DATA_BLOCK "PartErrorsCounter"   // DB46
{ S7_Optimized_Access := 'TRUE' }
VERSION : 0.1
// stored: AutoNumber true, DBAccessibleFromOPCUA true, DBAccessibleFromWebserver true, IsOnlyStoredInLoadMemory false, IsRetainMemResEnabled false, IsWriteProtectedInAS false, MemoryReserve 100
   VAR RETAIN
      CountersRef { S7_SetPoint := 'True'} : Array[1.."NumberOfProductionPrograms"] of "UDT_NOKcounter";
   END_VAR
   VAR
      CountersHMI : "UDT_NOKcounter";
   END_VAR
BEGIN
   CountersRef[1].Counters[0,0..50] := 0;
   CountersRef[1].Counters[1,0..9] := 0;
   CountersRef[1].Counters[1,10] := 2;
   CountersRef[1].Counters[1,11] := 1;
   CountersRef[1].Counters[1,12..19] := 0;
   CountersRef[1].Counters[1,20] := 3;
   CountersRef[1].Counters[1,21] := 1;
   CountersRef[1].Counters[1,22..33] := 0;
   CountersRef[1].Counters[1,34] := 1;
   CountersRef[1].Counters[1,35..43] := 0;
   CountersRef[1].Counters[1,44] := 1;
   CountersRef[1].Counters[1,45..50] := 0;
   CountersRef[1].Counters[2,0..13] := 0;
   CountersRef[1].Counters[2,14] := 1;
   CountersRef[1].Counters[2,15..20] := 0;
   CountersRef[1].Counters[2,21] := 1;
   CountersRef[1].Counters[2,22..50] := 0;
   CountersRef[1].Counters[3,0..50] := 0;
   CountersRef[2].Counters[0,0..50] := 0;
   CountersRef[2].Counters[1,0..9] := 0;
   CountersRef[2].Counters[1,10] := 4;
   CountersRef[2].Counters[1,11] := 1;
   CountersRef[2].Counters[1,12..19] := 0;
   CountersRef[2].Counters[1,20] := 3;
   CountersRef[2].Counters[1,21] := 2;
   CountersRef[2].Counters[1,22..50] := 0;
   CountersRef[2].Counters[2,0..10] := 0;
   CountersRef[2].Counters[2,11] := 1;
   CountersRef[2].Counters[2,12..13] := 0;
   CountersRef[2].Counters[2,14] := 1;
   CountersRef[2].Counters[2,15..20] := 0;
   CountersRef[2].Counters[2,21] := 1;
   CountersRef[2].Counters[2,22..23] := 0;
   CountersRef[2].Counters[2,24] := 1;
   CountersRef[2].Counters[2,25..30] := 0;
   CountersRef[2].Counters[2,31] := 1;
   CountersRef[2].Counters[2,32..33] := 0;
   CountersRef[2].Counters[2,34] := 1;
   CountersRef[2].Counters[2,35..40] := 0;
   CountersRef[2].Counters[2,41] := 1;
   CountersRef[2].Counters[2,42..43] := 0;
   CountersRef[2].Counters[2,44] := 1;
   CountersRef[2].Counters[2,45..50] := 0;
   CountersRef[2].Counters[3,0..50] := 0;
   CountersRef[3].Counters[0,0..50] := 0;
   CountersRef[3].Counters[1,0..50] := 0;
   CountersRef[3].Counters[2,0..50] := 0;
   CountersRef[3].Counters[3,0..50] := 0;
   CountersRef[4].Counters[0,0..50] := 0;
   CountersRef[4].Counters[1,0..50] := 0;
   CountersRef[4].Counters[2,0..50] := 0;
   CountersRef[4].Counters[3,0..50] := 0;
   CountersRef[5].Counters[0,0..50] := 0;
   CountersRef[5].Counters[1,0..9] := 0;
   CountersRef[5].Counters[1,10] := 17;
   CountersRef[5].Counters[1,11] := 6;
   CountersRef[5].Counters[1,12..19] := 0;
   CountersRef[5].Counters[1,20..21] := 1;
   CountersRef[5].Counters[1,22..50] := 0;
   CountersRef[5].Counters[2,0..9] := 0;
   CountersRef[5].Counters[2,10] := 4;
   CountersRef[5].Counters[2,11] := 3;
   CountersRef[5].Counters[2,12..13] := 0;
   CountersRef[5].Counters[2,14] := 1;
   CountersRef[5].Counters[2,15..23] := 0;
   CountersRef[5].Counters[2,24] := 4;
   CountersRef[5].Counters[2,25..50] := 0;
   CountersRef[5].Counters[3,0..50] := 0;
   CountersRef[6].Counters[0,0..50] := 0;
   CountersRef[6].Counters[1,0..50] := 0;
   CountersRef[6].Counters[2,0..9] := 0;
   CountersRef[6].Counters[2,10] := 1;
   CountersRef[6].Counters[2,11..13] := 0;
   CountersRef[6].Counters[2,14] := 1;
   CountersRef[6].Counters[2,15..21] := 0;
   CountersRef[6].Counters[2,22] := 1;
   CountersRef[6].Counters[2,23..33] := 0;
   CountersRef[6].Counters[2,34] := 2;
   CountersRef[6].Counters[2,35..43] := 0;
   CountersRef[6].Counters[2,44] := 2;
   CountersRef[6].Counters[2,45..50] := 0;
   CountersRef[6].Counters[3,0..50] := 0;
   CountersRef[7].Counters[0,0..50] := 0;
   CountersRef[7].Counters[1,0..50] := 0;
   CountersRef[7].Counters[2,0..50] := 0;
   CountersRef[7].Counters[3,0..50] := 0;
   CountersRef[8].Counters[0,0..50] := 0;
   CountersRef[8].Counters[1,0..50] := 0;
   CountersRef[8].Counters[2,0..50] := 0;
   CountersRef[8].Counters[3,0..50] := 0;
   CountersHMI.Counters[0,0..50] := 0;
   CountersHMI.Counters[1,0..50] := 0;
   CountersHMI.Counters[2,0..50] := 0;
   CountersHMI.Counters[3,0..50] := 0;
END_DATA_BLOCK

DATA_BLOCK "READER_MODEL"   // DB74
{ S7_Optimized_Access := 'TRUE' }
VERSION : 0.1
// stored: AutoNumber true, DBAccessibleFromOPCUA true, DBAccessibleFromWebserver true, IsOnlyStoredInLoadMemory false, IsRetainMemResEnabled false, IsWriteProtectedInAS false, MemoryReserve 100
   VAR RETAIN
      PRODUCT { S7_SetPoint := 'True'} : Array[0.."NumberOfProductionPrograms"] of "READER_PRODUCT";
   END_VAR
BEGIN
   PRODUCT[1..4].SIDE_RH.POSITION := 13;
   PRODUCT[1..4].SIDE_RH.LEN := 3;
   PRODUCT[1].SIDE_RH.STRING_LABEL := '336';
   PRODUCT[2].SIDE_RH.STRING_LABEL := '532';
   PRODUCT[3].SIDE_RH.STRING_LABEL := '336';
   PRODUCT[4].SIDE_RH.STRING_LABEL := '532';
   PRODUCT[1..4].SIDE_RH.READER_BYPASS := FALSE;
   PRODUCT[1..4].SIDE_LH.POSITION := 13;
   PRODUCT[1..4].SIDE_LH.LEN := 3;
   PRODUCT[1].SIDE_LH.STRING_LABEL := '328';
   PRODUCT[2].SIDE_LH.STRING_LABEL := '526';
   PRODUCT[3].SIDE_LH.STRING_LABEL := '328';
   PRODUCT[4].SIDE_LH.STRING_LABEL := '526';
   PRODUCT[1..4].SIDE_LH.READER_BYPASS := FALSE;
   PRODUCT[1..4].REAR_TUBE.POSITION := 13;
   PRODUCT[1..4].REAR_TUBE.LEN := 3;
   PRODUCT[1].REAR_TUBE.STRING_LABEL := '343';
   PRODUCT[2].REAR_TUBE.STRING_LABEL := '514';
   PRODUCT[3].REAR_TUBE.STRING_LABEL := '343';
   PRODUCT[4].REAR_TUBE.STRING_LABEL := '514';
   PRODUCT[1..4].REAR_TUBE.READER_BYPASS := FALSE;
   PRODUCT[1..2].FRONT_TUBE.POSITION := 13;
   PRODUCT[1..2].FRONT_TUBE.LEN := 3;
   PRODUCT[1..2].FRONT_TUBE.STRING_LABEL := '907';
   PRODUCT[1..4].FRONT_TUBE.READER_BYPASS := TRUE;
   PRODUCT[1..2].NUM_TUBE := TRUE;
   PRODUCT[3].NUM_TUBE := FALSE;
END_DATA_BLOCK

DATA_BLOCK "READER_MODEL_ACTUAL"   // DB75
{ S7_Optimized_Access := 'TRUE' }
VERSION : 0.1
// stored: AutoNumber true, DBAccessibleFromOPCUA true, DBAccessibleFromWebserver true, IsOnlyStoredInLoadMemory false, IsRetainMemResEnabled false, IsWriteProtectedInAS false, MemoryReserve 100
   VAR
      PRODUCTO : "READER_PRODUCT";
      ST1_TABLE_1 : Struct
         SIDE_RH : String;
         SIDE_LH : String;
         REAR_TUBE : String;
         FRONT_TUBE : String;
         NFP_AUX : String;
      END_STRUCT;
      ST2_TABLE_2 : Struct
         SIDE_RH : String;
         SIDE_LH : String;
         REAR_TUBE : String;
         FRONT_TUBE : String;
         NFP_AUX : String;
      END_STRUCT;
      ST3_FITTING : Struct
         SIDE_RH : String;
         SIDE_LH : String;
         REAR_TUBE : String;
         FRONT_TUBE : String;
         NFP_AUX : String;
      END_STRUCT;
      R1_GRIPPER : Struct
         SIDE_RH : String;
         SIDE_LH : String;
         REAR_TUBE : String;
         FRONT_TUBE : String;
         NFP_AUX : String;
      END_STRUCT;
      R2_GRIPPER : Struct
         SIDE_RH : String;
         SIDE_LH : String;
         REAR_TUBE : String;
         FRONT_TUBE : String;
         NFP_AUX : String;
      END_STRUCT;
      ALL_SCANNER_OK : Bool;
      SIDE_LH_SCANNER_OK : Bool;
      SIDE_RH_SCANNER_OK : Bool;
      REAR_TUBE_SCANNER_OK : Bool;
      FRONT_TUBE_SCANNER_OK : Bool;
      IN_BOX : "READER_PRODUCT";
      EDIT : "READER_PRODUCT";
      READER { S7_SetPoint := 'True'} : String;
      ST_CLEAR : Struct
         SIDE_RH : String;
         SIDE_LH : String;
         REAR_TUBE : String;
         FRONT_TUBE : String;
         NFP_AUX : String;
      END_STRUCT;
      SCAN_CLEAR : Bool;
      RECIBIDO_ESCANER_REAR_TUBE : Array[0..254] of Char;
      RECIBIDO_ESCANER_FRONT_TUBE : Array[0..254] of Char;
      RECIBIDO_ESCANER_RH_MEMBER : Array[0..254] of Char;
      RECIBIDO_ESCANER_LH_MEMBER : Array[0..254] of Char;
      RECIBIDO_ESCANER_REAR_TUBE_STRING : String;
      RECIBIDO_ESCANER_FRONT_TUBE_STRING : String;
      RECIBIDO_ESCANER_RH_MEMBER_STRING : String;
      RECIBIDO_ESCANER_LH_MEMBER_STRING : String;
      LECTURA_ESCANER_REAR_TUBE : String;
      LECTURA_ESCANER_FRONT_TUBE : String;
      LECTURA_ESCANER_RH_MEMBER : String;
      LECTURA_ESCANER_LH_MEMBER : String;
   END_VAR
BEGIN
END_DATA_BLOCK

DATA_BLOCK "MII_Interface_Configuration"   // DB2021
{ S7_Optimized_Access := 'TRUE' }
VERSION : 0.1
// stored: AutoNumber false, DBAccessibleFromOPCUA true, DBAccessibleFromWebserver true, IsOnlyStoredInLoadMemory false, IsRetainMemResEnabled false, IsWriteProtectedInAS false, MemoryReserve 100
   VAR
      Connection { ExternalAccessible := 'False'; ExternalVisible := 'False'; ExternalWritable := 'False'} : Struct
         ConnectInfo { ExternalAccessible := 'False'; ExternalVisible := 'False'; ExternalWritable := 'False'; S7_SetPoint := 'True'} : OPC_UA_SessionConnectInfo;
         ConnectionHdl { ExternalAccessible := 'False'; ExternalVisible := 'False'; ExternalWritable := 'False'} : DWord;
         ServerEndpointUrl { ExternalAccessible := 'False'; ExternalVisible := 'False'; ExternalWritable := 'False'} : String[254] := 'opc.tcp://:4840';
      END_STRUCT;
      Namespaces { ExternalAccessible := 'False'; ExternalVisible := 'False'; ExternalWritable := 'False'} : Struct
         NamespaceURIs { ExternalAccessible := 'False'; ExternalVisible := 'False'; ExternalWritable := 'False'} : Array[0..0] of WString;
         ServerNamespaceIndexes { ExternalAccessible := 'False'; ExternalVisible := 'False'; ExternalWritable := 'False'} : Array[0..0] of UInt;
         NamespaceStatusList { ExternalAccessible := 'False'; ExternalVisible := 'False'; ExternalWritable := 'False'} : Array[0..0] of DWord;
         NamespaceCount { ExternalAccessible := 'False'; ExternalVisible := 'False'; ExternalWritable := 'False'} : UInt := 1;
      END_STRUCT;
      MethodLists { ExternalAccessible := 'False'; ExternalVisible := 'False'; ExternalWritable := 'False'} : Struct
         MII_METHODS { ExternalAccessible := 'False'; ExternalVisible := 'False'; ExternalWritable := 'False'} : Struct
            MethodCount { ExternalAccessible := 'False'; ExternalVisible := 'False'; ExternalWritable := 'False'} : UInt := 9;
            ObjectNodes { ExternalAccessible := 'False'; ExternalVisible := 'False'; ExternalWritable := 'False'; S7_SetPoint := 'True'} : Array[0..8] of OPC_UA_NodeId;
            MethodNodes { ExternalAccessible := 'False'; ExternalVisible := 'False'; ExternalWritable := 'False'; S7_SetPoint := 'True'} : Array[0..8] of OPC_UA_NodeId;
            MethodHdls { ExternalAccessible := 'False'; ExternalVisible := 'False'; ExternalWritable := 'False'} : Array[0..8] of DWord;
         END_STRUCT;
      END_STRUCT;
   END_VAR
BEGIN
   Connection.ConnectInfo.SessionName := WSTRING#'OPC UA Connection_1';
   Connection.ConnectInfo.ApplicationName := WSTRING#'';
   Connection.ConnectInfo.SecurityMsgMode := 1;
   Connection.ConnectInfo.SecurityPolicy := 1;
   Connection.ConnectInfo.CheckServerCertificate := False;
   Connection.ConnectInfo.TransportProfile := 1;
   Connection.ConnectInfo.UserIdentityTokenType := 0;
   Connection.ConnectInfo.CertificateID := 0;
   Connection.ConnectInfo.SessionTimeout := T#30S;
   Connection.ConnectInfo.MonitorConnection := T#5S;
   Connection.ConnectInfo.LocaleIDs[0] := 'en-US';
   Connection.ConnectInfo.LocaleIDs[1..4] := '';
   Namespaces.NamespaceURIs[0] := WSTRING#'http://sap.com/PCoUaServer/Destinations';
   MethodLists.MII_METHODS.ObjectNodes[0..8].NamespaceIndex := 0;
   MethodLists.MII_METHODS.ObjectNodes[0..8].Identifier := WSTRING#'a72e725d-6be7-4a17-bcd4-0be67b6cbfbe';
   MethodLists.MII_METHODS.ObjectNodes[0..8].IdentifierType := 1;
   MethodLists.MII_METHODS.MethodNodes[0..8].NamespaceIndex := 0;
   MethodLists.MII_METHODS.MethodNodes[0].Identifier := WSTRING#'5e83d9d8-abe4-4ece-894f-119f40c23d1f';
   MethodLists.MII_METHODS.MethodNodes[1].Identifier := WSTRING#'3a6a30a3-a9b9-4f00-ac48-5dfb28f8e6a4';
   MethodLists.MII_METHODS.MethodNodes[2].Identifier := WSTRING#'fc62dbc1-f795-4566-bb4d-0b596c22b389';
   MethodLists.MII_METHODS.MethodNodes[3].Identifier := WSTRING#'c66a08a9-d6b4-453f-b0e9-0d4ff2f595c1';
   MethodLists.MII_METHODS.MethodNodes[4].Identifier := WSTRING#'a12cda35-f7c0-4943-b30d-d26694925508';
   MethodLists.MII_METHODS.MethodNodes[5].Identifier := WSTRING#'9febe458-2cc0-4c91-b17b-56067f98920d';
   MethodLists.MII_METHODS.MethodNodes[6].Identifier := WSTRING#'9fd0466f-1121-4821-944e-2d89fa189b19';
   MethodLists.MII_METHODS.MethodNodes[7].Identifier := WSTRING#'1a97343a-fec3-434f-bd32-25d77a49b705';
   MethodLists.MII_METHODS.MethodNodes[8].Identifier := WSTRING#'d0a2f4c1-2dea-442d-aa14-aa44dfe57828';
   MethodLists.MII_METHODS.MethodNodes[0..8].IdentifierType := 1;
END_DATA_BLOCK

DATA_BLOCK "MII_Interface_Data"   // DB2022
{ S7_Optimized_Access := 'TRUE' }
VERSION : 0.1
// stored: AutoNumber false, DBAccessibleFromOPCUA true, DBAccessibleFromWebserver true, IsOnlyStoredInLoadMemory false, IsRetainMemResEnabled false, IsWriteProtectedInAS false, MemoryReserve 100
   VAR
      MII_METHODS { ExternalAccessible := 'False'; ExternalVisible := 'False'; ExternalWritable := 'False'} : Struct
         MethodStatusList { ExternalAccessible := 'False'; ExternalVisible := 'False'; ExternalWritable := 'False'} : Array[0..8] of DWord;
         MethodResultList { ExternalAccessible := 'False'; ExternalVisible := 'False'; ExternalWritable := 'False'} : Array[0..8] of DWord;
         M000_PRODUCTION_DECLARATION { ExternalAccessible := 'False'; ExternalVisible := 'False'; ExternalWritable := 'False'} : Struct
            Inputs { ExternalAccessible := 'False'; ExternalVisible := 'False'; ExternalWritable := 'False'; S7_SetPoint := 'True'} : "MII_Interface.MII_METHODS.M000_PRODUCTION_DECLARATION.Inputs";   // the definition of the input argument of method 1:Destinations.1:PRODUCTION_DECLARATION
            Outputs { ExternalAccessible := 'False'; ExternalVisible := 'False'; ExternalWritable := 'False'; S7_SetPoint := 'True'} : "MII_Interface.MII_METHODS.M000_PRODUCTION_DECLARATION.Outputs";   // the definition of the output arguments of method 1:Destinations.1:PRODUCTION_DECLARATION
         END_STRUCT;
         M001_GET_LOCAL_TIME { ExternalAccessible := 'False'; ExternalVisible := 'False'; ExternalWritable := 'False'} : Struct
            Outputs { ExternalAccessible := 'False'; ExternalVisible := 'False'; ExternalWritable := 'False'; S7_SetPoint := 'True'} : "MII_Interface.MII_METHODS.M001_GET_LOCAL_TIME.Outputs";   // the definition of the output arguments of method 2:Destinations.2:2_GET_LOCAL_TIME
         END_STRUCT;
         M101_SCRAP_DECLARATION { ExternalAccessible := 'False'; ExternalVisible := 'False'; ExternalWritable := 'False'} : Struct
            Inputs { ExternalAccessible := 'False'; ExternalVisible := 'False'; ExternalWritable := 'False'; S7_SetPoint := 'True'} : "MII_Interface.MII_METHODS.M101_SCRAP_DECLARATION.Inputs";   // the definition of the input argument of method 2:Destinations.2:1_SCRAP_DECLARATION
            Outputs { ExternalAccessible := 'False'; ExternalVisible := 'False'; ExternalWritable := 'False'; S7_SetPoint := 'True'} : "MII_Interface.MII_METHODS.M101_SCRAP_DECLARATION.Outputs";   // the definition of the output arguments of method 2:Destinations.2:1_SCRAP_DECLARATION
         END_STRUCT;
         M003_GENERATE_ALERT { ExternalAccessible := 'False'; ExternalVisible := 'False'; ExternalWritable := 'False'} : Struct
            Inputs { ExternalAccessible := 'False'; ExternalVisible := 'False'; ExternalWritable := 'False'; S7_SetPoint := 'True'} : "MII_Interface.MII_METHODS.M003_GENERATE_ALERT.Inputs";   // the definition of the input argument of method 2:Destinations.2:3_GENERATE_ALERT
            Outputs { ExternalAccessible := 'False'; ExternalVisible := 'False'; ExternalWritable := 'False'; S7_SetPoint := 'True'} : "MII_Interface.MII_METHODS.M003_GENERATE_ALERT.Outputs";   // the definition of the output arguments of method 2:Destinations.2:3_GENERATE_ALERT
         END_STRUCT;
         M102_REWORK_DECLARATION { ExternalAccessible := 'False'; ExternalVisible := 'False'; ExternalWritable := 'False'} : Struct
            Inputs { ExternalAccessible := 'False'; ExternalVisible := 'False'; ExternalWritable := 'False'; S7_SetPoint := 'True'} : "MII_Interface.MII_METHODS.M102_REWORK_DECLARATION.Inputs";   // the definition of the input argument of method 2:Destinations.2:4_REWORK_DECLARATION
            Outputs { ExternalAccessible := 'False'; ExternalVisible := 'False'; ExternalWritable := 'False'; S7_SetPoint := 'True'} : "MII_Interface.MII_METHODS.M102_REWORK_DECLARATION.Outputs";   // the definition of the output arguments of method 2:Destinations.2:4_REWORK_DECLARATION
         END_STRUCT;
         M002_GET_PLANTS { ExternalAccessible := 'False'; ExternalVisible := 'False'; ExternalWritable := 'False'} : Struct
            Outputs { ExternalAccessible := 'False'; ExternalVisible := 'False'; ExternalWritable := 'False'; S7_SetPoint := 'True'} : "MII_Interface.MII_METHODS.M002_GET_PLANTS.Outputs";   // the definition of the output arguments of method 2:Destinations.2:M005_GET_PLANTS
         END_STRUCT;
         M004_NTRS { ExternalAccessible := 'False'; ExternalVisible := 'False'; ExternalWritable := 'False'} : Struct
            Inputs { ExternalAccessible := 'False'; ExternalVisible := 'False'; ExternalWritable := 'False'; S7_SetPoint := 'True'} : "MII_Interface.MII_METHODS.M004_NTRS.Inputs";   // the definition of the input argument of method 2:Destinations.2:M006_NTRS
            Outputs { ExternalAccessible := 'False'; ExternalVisible := 'False'; ExternalWritable := 'False'; S7_SetPoint := 'True'} : "MII_Interface.MII_METHODS.M004_NTRS.Outputs";   // the definition of the output arguments of method 2:Destinations.2:M006_NTRS
         END_STRUCT;
         M103_PY { ExternalAccessible := 'False'; ExternalVisible := 'False'; ExternalWritable := 'False'} : Struct
            Inputs { ExternalAccessible := 'False'; ExternalVisible := 'False'; ExternalWritable := 'False'; S7_SetPoint := 'True'} : "MII_Interface.MII_METHODS.M103_PY.Inputs";   // the definition of the input argument of method 2:Destinations.2:M103_PY
            Outputs { ExternalAccessible := 'False'; ExternalVisible := 'False'; ExternalWritable := 'False'; S7_SetPoint := 'True'} : "MII_Interface.MII_METHODS.M103_PY.Outputs";   // the definition of the output arguments of method 2:Destinations.2:M103_PY
         END_STRUCT;
         M005_VARIABILITY { ExternalAccessible := 'False'; ExternalVisible := 'False'; ExternalWritable := 'False'} : Struct
            Inputs { ExternalAccessible := 'False'; ExternalVisible := 'False'; ExternalWritable := 'False'; S7_SetPoint := 'True'} : "MII_Interface.MII_METHODS.M005_VARIABILITY.Inputs";   // the definition of the input argument of method 2:Destinations.2:M005_VARIABILITY
            Outputs { ExternalAccessible := 'False'; ExternalVisible := 'False'; ExternalWritable := 'False'; S7_SetPoint := 'True'} : "MII_Interface.MII_METHODS.M005_VARIABILITY.Outputs";   // the definition of the output arguments of method 2:Destinations.2:M005_VARIABILITY
         END_STRUCT;
      END_STRUCT;
   END_VAR
BEGIN
END_DATA_BLOCK

ORGANIZATION_BLOCK "OB_ProgramCycle"   // OB1, LAD, ProgramCycle
TITLE = "Main Program Sweep (Cycle)"
{ S7_Optimized_Access := 'TRUE' }
VERSION : 0.1
// stored: AutoNumber true, IsIECCheckEnabled false, SetENOAutomatically false
   VAR_INPUT
      Initial_Call : Bool;   // Initial call of this OB
      Remanence : Bool;   // =True, if remanent data are available
   END_VAR
   VAR_TEMP   // added for the SCL form of the ladder/FBD networks
      _w1 : Bool;
      _s5time1 : S5Time;
   END_VAR
BEGIN

REGION Network 1
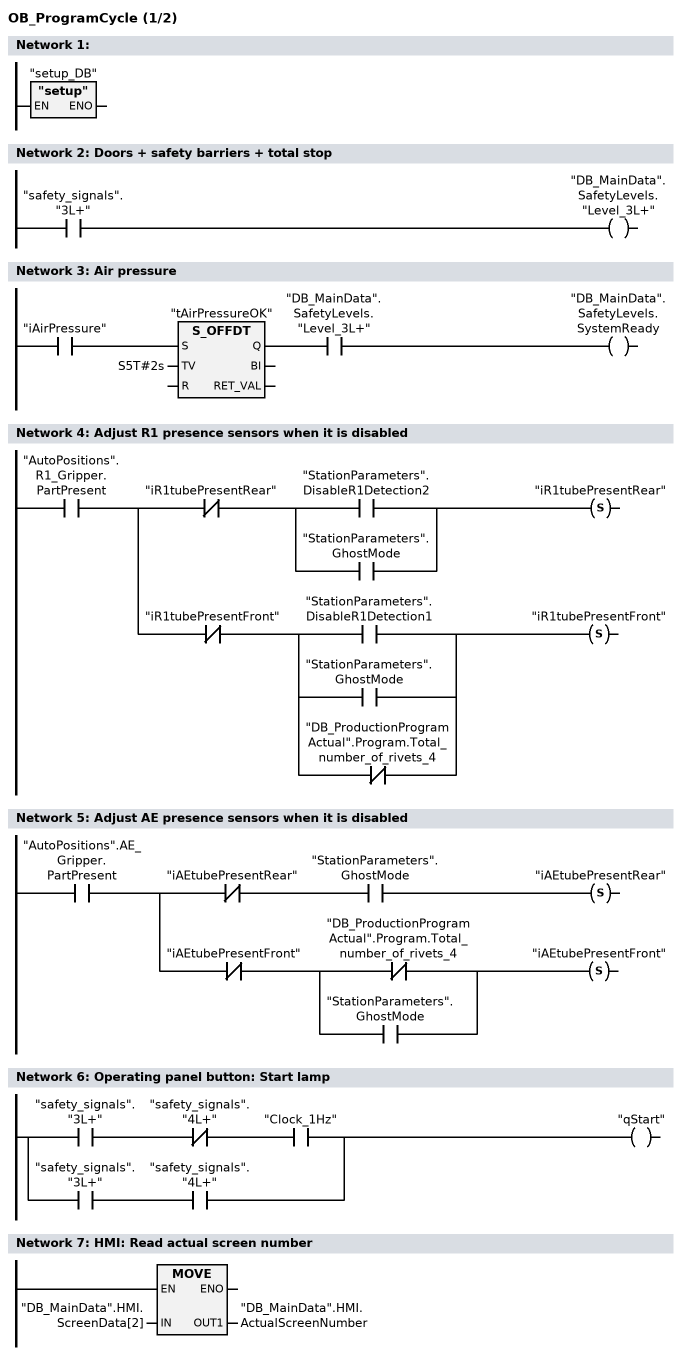
   RUNG wire#powerrail
      "setup_DB"()
   END_RUNG
   // the same network as SCL:
   "setup_DB"();   // "setup"
END_REGION

REGION Network 2: Doors + safety barriers + total stop
   RUNG wire#powerrail
      Contact( "safety_signals"."3L+" )
      Coil( "DB_MainData".SafetyLevels."Level_3L+" )
   END_RUNG
   // the same network as SCL:
   "DB_MainData".SafetyLevels."Level_3L+" := "safety_signals"."3L+";
END_REGION

REGION Network 3: Air pressure
   RUNG wire#powerrail
      Contact( "iAirPressure" )
      S_OFFDT(T_NO := "tAirPressureOK", TV := S5T#2s, R :=, BI =>, RET_VAL =>)
      Contact( "DB_MainData".SafetyLevels."Level_3L+" )
      Coil( "DB_MainData".SafetyLevels.SystemReady )
   END_RUNG
   // the same network as SCL:
   #_s5time1 := S_OFFDT(T_NO := "tAirPressureOK", S := "iAirPressure", TV := S5T#2s, Q => #_w1);
   "DB_MainData".SafetyLevels.SystemReady := #_w1 AND "DB_MainData".SafetyLevels."Level_3L+";
END_REGION

REGION Network 4: Adjust R1 presence sensors when it is disabled
   RUNG wire#powerrail
      Contact( "AutoPositions".R1_Gripper.PartPresent )
      wire#w1
      I_Contact( "iR1tubePresentRear" )
      wire#w2
      Contact( "StationParameters".DisableR1Detection2 )
      wire#w3
      S_Coil( "iR1tubePresentRear" )
   END_RUNG
   RUNG wire#w2
      Contact( "StationParameters".GhostMode )
   END_RUNG wire#w3
   RUNG wire#w1
      I_Contact( "iR1tubePresentFront" )
      wire#w4
      Contact( "StationParameters".DisableR1Detection1 )
      wire#w5
      S_Coil( "iR1tubePresentFront" )
   END_RUNG
   RUNG wire#w4
      Contact( "StationParameters".GhostMode )
   END_RUNG wire#w5
   RUNG wire#w4
      I_Contact( "DB_ProductionProgramActual".Program.Total_number_of_rivets_4 )
   END_RUNG wire#w5
   // the same network as SCL:
   IF "AutoPositions".R1_Gripper.PartPresent AND NOT "iR1tubePresentRear" AND ("StationParameters".DisableR1Detection2 OR "StationParameters".GhostMode) THEN
       "iR1tubePresentRear" := TRUE;
   END_IF;
   IF "AutoPositions".R1_Gripper.PartPresent AND NOT "iR1tubePresentFront" AND ("StationParameters".DisableR1Detection1 OR "StationParameters".GhostMode OR NOT "DB_ProductionProgramActual".Program.Total_number_of_rivets_4) THEN
       "iR1tubePresentFront" := TRUE;
   END_IF;
END_REGION

REGION Network 5: Adjust AE presence sensors when it is disabled
   RUNG wire#powerrail
      Contact( "AutoPositions".AE_Gripper.PartPresent )
      wire#w1
      I_Contact( "iAEtubePresentRear" )
      Contact( "StationParameters".GhostMode )
      S_Coil( "iAEtubePresentRear" )
   END_RUNG
   RUNG wire#w1
      I_Contact( "iAEtubePresentFront" )
      wire#w2
      I_Contact( "DB_ProductionProgramActual".Program.Total_number_of_rivets_4 )
      wire#w3
      S_Coil( "iAEtubePresentFront" )
   END_RUNG
   RUNG wire#w2
      Contact( "StationParameters".GhostMode )
   END_RUNG wire#w3
   // the same network as SCL:
   IF "AutoPositions".AE_Gripper.PartPresent AND NOT "iAEtubePresentRear" AND "StationParameters".GhostMode THEN
       "iAEtubePresentRear" := TRUE;
   END_IF;
   IF "AutoPositions".AE_Gripper.PartPresent AND NOT "iAEtubePresentFront" AND (NOT "DB_ProductionProgramActual".Program.Total_number_of_rivets_4 OR "StationParameters".GhostMode) THEN
       "iAEtubePresentFront" := TRUE;
   END_IF;
END_REGION

REGION Network 6: Operating panel button: Start lamp
   RUNG wire#powerrail
      Contact( "safety_signals"."3L+" )
      I_Contact( "safety_signals"."4L+" )
      Contact( "Clock_1Hz" )
      wire#w1
      Coil( "qStart" )
   END_RUNG
   RUNG wire#powerrail
      Contact( "safety_signals"."3L+" )
      Contact( "safety_signals"."4L+" )
   END_RUNG wire#w1
   // the same network as SCL:
   "qStart" := ("safety_signals"."3L+" AND NOT "safety_signals"."4L+" AND "Clock_1Hz") OR ("safety_signals"."3L+" AND "safety_signals"."4L+");
END_REGION

REGION Network 7: HMI: Read actual screen number
   RUNG wire#powerrail
      Move(in := "DB_MainData".HMI.ScreenData[2], out1 => "DB_MainData".HMI.ActualScreenNumber)
   END_RUNG
   // the same network as SCL:
   "DB_MainData".HMI.ActualScreenNumber := "DB_MainData".HMI.ScreenData[2];
END_REGION

REGION Network 8: FB_Main
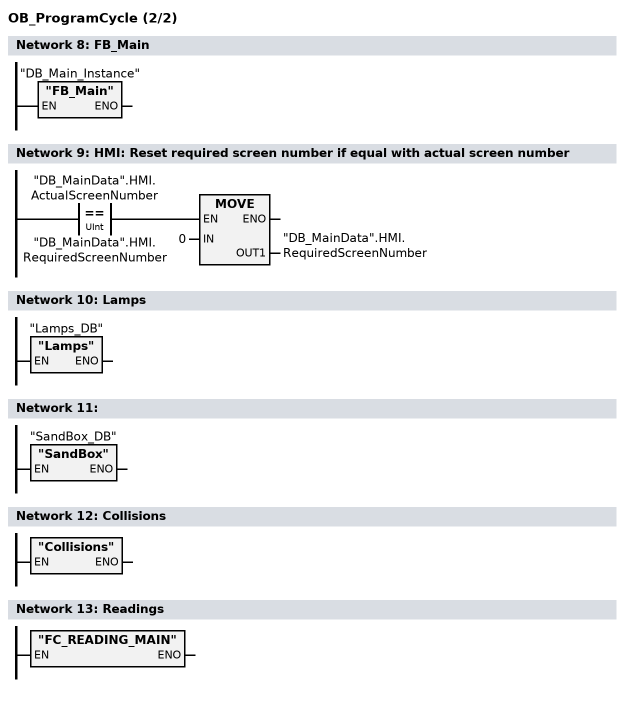
   RUNG wire#powerrail
      "DB_Main_Instance"()
   END_RUNG
   // the same network as SCL:
   "DB_Main_Instance"();   // "FB_Main"
END_REGION

REGION Network 9: HMI: Reset required screen number if equal with actual screen number
   RUNG wire#powerrail
      { S7_Templates := "SrcType := UInt" } EQ_Contact(in1 := "DB_MainData".HMI.ActualScreenNumber, in2 := "DB_MainData".HMI.RequiredScreenNumber)
      Move(in := 0, out1 => "DB_MainData".HMI.RequiredScreenNumber)
   END_RUNG
   // the same network as SCL:
   IF "DB_MainData".HMI.ActualScreenNumber = "DB_MainData".HMI.RequiredScreenNumber THEN
       "DB_MainData".HMI.RequiredScreenNumber := 0;
   END_IF;
END_REGION

REGION Network 10: Lamps
   RUNG wire#powerrail
      "Lamps_DB"()
   END_RUNG
   // the same network as SCL:
   "Lamps_DB"();   // "Lamps"
END_REGION

REGION Network 11
   RUNG wire#powerrail
      "SandBox_DB"()
   END_RUNG
   // the same network as SCL:
   "SandBox_DB"();   // "SandBox"
END_REGION

REGION Network 12: Collisions
   RUNG wire#powerrail
      "Collisions"()
   END_RUNG
   // the same network as SCL:
   "Collisions"();
END_REGION

REGION Network 13: Readings
   RUNG wire#powerrail
      "FC_READING_MAIN"()
   END_RUNG
   // the same network as SCL:
   "FC_READING_MAIN"();
END_REGION
END_ORGANIZATION_BLOCK

FUNCTION_BLOCK "FB_Main"   // FB5000, LAD
{ S7_Optimized_Access := 'TRUE' }
VERSION : 0.1
// stored: AutoNumber false, IsIECCheckEnabled false, IsRetainMemResEnabled false, MemoryReserve 100, SetENOAutomatically false, UDAEnableTagReadback false
   VAR
      IEC_Timer_0_Instance { S7_SetPoint := 'True'} : TON_TIME;
      MachineModeOld { S7_SetPoint := 'True'} : UInt;
      F_TRIG_Instance { S7_SetPoint := 'True'} : F_TRIG;
      F_TRIG_Instance_1 { S7_SetPoint := 'True'} : F_TRIG;
      F_TRIG_Instance_2 { S7_SetPoint := 'True'} : F_TRIG;
      R_TRIG_Instance { S7_SetPoint := 'True'} : R_TRIG;
      R_TRIG_Instance_1 { S7_SetPoint := 'True'} : R_TRIG;
   END_VAR
   VAR_TEMP   // added for the SCL form of the ladder/FBD networks
      _w1 : Bool;
      _w2 : Bool;
   END_VAR
BEGIN

REGION Network 1: alarms fc, lamp fc
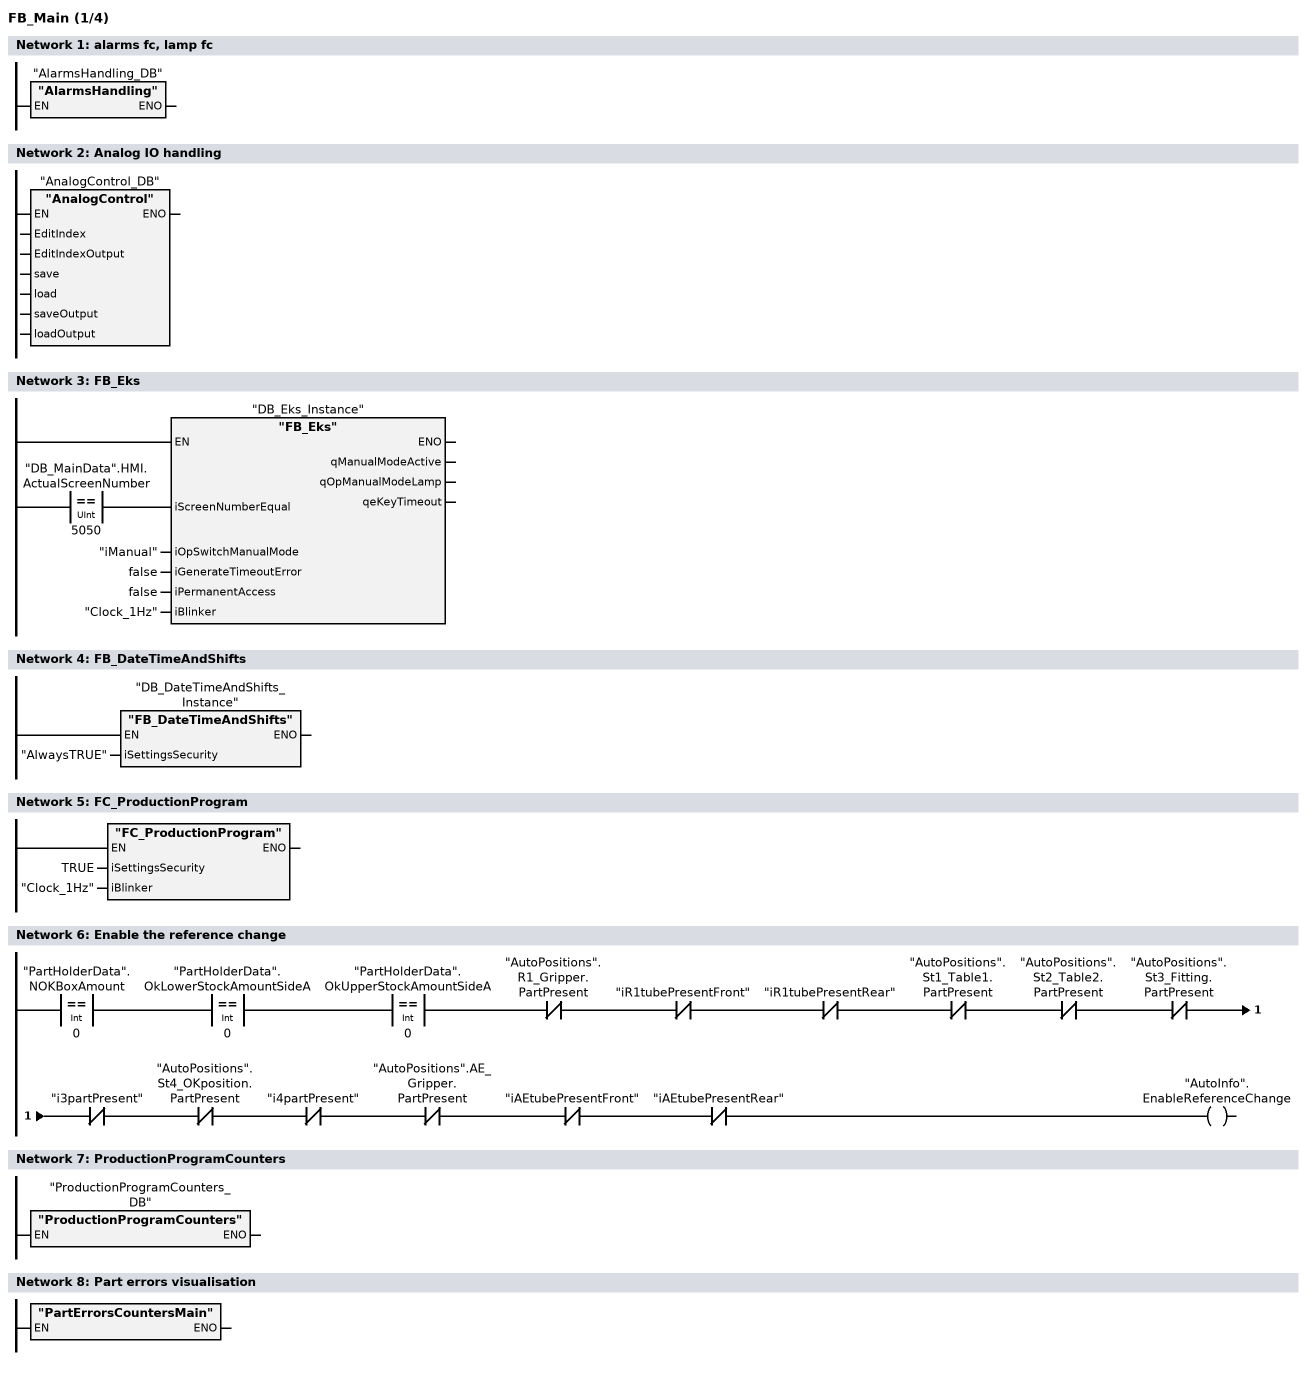
   RUNG wire#powerrail
      "AlarmsHandling_DB"()
   END_RUNG
   // the same network as SCL:
   "AlarmsHandling_DB"();   // "AlarmsHandling"
END_REGION

REGION Network 2: Analog IO handling
   RUNG wire#powerrail
      "AnalogControl_DB"(EditIndex :=, save :=, load :=, EditIndexOutput :=, saveOutput :=, loadOutput :=)
   END_RUNG
   // the same network as SCL:
   "AnalogControl_DB"();   // "AnalogControl"
END_REGION

REGION Network 3: FB_Eks
   RUNG wire#powerrail
      "DB_Eks_Instance"(iScreenNumberEqual := wire#w1, iOpSwitchManualMode := "iManual", iGenerateTimeoutError := false, iPermanentAccess := false, iBlinker := "Clock_1Hz", qManualModeActive =>, qOpManualModeLamp =>, qeKeyTimeout =>)
   END_RUNG
   RUNG wire#powerrail
      { S7_Templates := "SrcType := UInt" } EQ_Contact(in1 := "DB_MainData".HMI.ActualScreenNumber, in2 := 5050)
   END_RUNG wire#w1
   // the same network as SCL:
   "DB_Eks_Instance"(iScreenNumberEqual := "DB_MainData".HMI.ActualScreenNumber = 5050,   // "FB_Eks"
                     iOpSwitchManualMode := "iManual",
                     iGenerateTimeoutError := false,
                     iPermanentAccess := false,
                     iBlinker := "Clock_1Hz");
END_REGION

REGION Network 4: FB_DateTimeAndShifts
   RUNG wire#powerrail
      "DB_DateTimeAndShifts_Instance"(iSettingsSecurity := "AlwaysTRUE")
   END_RUNG
   // the same network as SCL:
   "DB_DateTimeAndShifts_Instance"(iSettingsSecurity := "AlwaysTRUE");   // "FB_DateTimeAndShifts"
END_REGION

REGION Network 5: FC_ProductionProgram
   RUNG wire#powerrail
      "FC_ProductionProgram"(iSettingsSecurity := TRUE, iBlinker := "Clock_1Hz")
   END_RUNG
   // the same network as SCL:
   "FC_ProductionProgram"(iSettingsSecurity := TRUE, iBlinker := "Clock_1Hz");
END_REGION

REGION Network 6: Enable the reference change
   RUNG wire#powerrail
      { S7_Templates := "SrcType := Int" } EQ_Contact(in1 := "PartHolderData".NOKBoxAmount, in2 := 0)
      { S7_Templates := "SrcType := Int" } EQ_Contact(in1 := "PartHolderData".OkLowerStockAmountSideA, in2 := 0)
      { S7_Templates := "SrcType := Int" } EQ_Contact(in1 := "PartHolderData".OkUpperStockAmountSideA, in2 := 0)
      I_Contact( "AutoPositions".R1_Gripper.PartPresent )
      I_Contact( "iR1tubePresentFront" )
      I_Contact( "iR1tubePresentRear" )
      I_Contact( "AutoPositions".St1_Table1.PartPresent )
      I_Contact( "AutoPositions".St2_Table2.PartPresent )
      I_Contact( "AutoPositions".St3_Fitting.PartPresent )
      I_Contact( "i3partPresent" )
      I_Contact( "AutoPositions".St4_OKposition.PartPresent )
      I_Contact( "i4partPresent" )
      I_Contact( "AutoPositions".AE_Gripper.PartPresent )
      I_Contact( "iAEtubePresentFront" )
      I_Contact( "iAEtubePresentRear" )
      Coil( "AutoInfo".EnableReferenceChange )
   END_RUNG
   // the same network as SCL:
   "AutoInfo".EnableReferenceChange := ("PartHolderData".NOKBoxAmount = 0) AND ("PartHolderData".OkLowerStockAmountSideA = 0) AND ("PartHolderData".OkUpperStockAmountSideA = 0) AND NOT "AutoPositions".R1_Gripper.PartPresent AND NOT "iR1tubePresentFront" AND NOT "iR1tubePresentRear" AND NOT "AutoPositions".St1_Table1.PartPresent AND NOT "AutoPositions".St2_Table2.PartPresent AND NOT "AutoPositions".St3_Fitting.PartPresent AND NOT "i3partPresent" AND NOT "AutoPositions".St4_OKposition.PartPresent AND NOT "i4partPresent" AND NOT "AutoPositions".AE_Gripper.PartPresent AND NOT "iAEtubePresentFront" AND NOT "iAEtubePresentRear";
END_REGION

REGION Network 7: ProductionProgramCounters
   RUNG wire#powerrail
      "ProductionProgramCounters_DB"()
   END_RUNG
   // the same network as SCL:
   "ProductionProgramCounters_DB"();   // "ProductionProgramCounters"
END_REGION

REGION Network 8: Part errors visualisation
   RUNG wire#powerrail
      "PartErrorsCountersMain"()
   END_RUNG
   // the same network as SCL:
   "PartErrorsCountersMain"();
END_REGION

REGION Network 9: FB_Devices
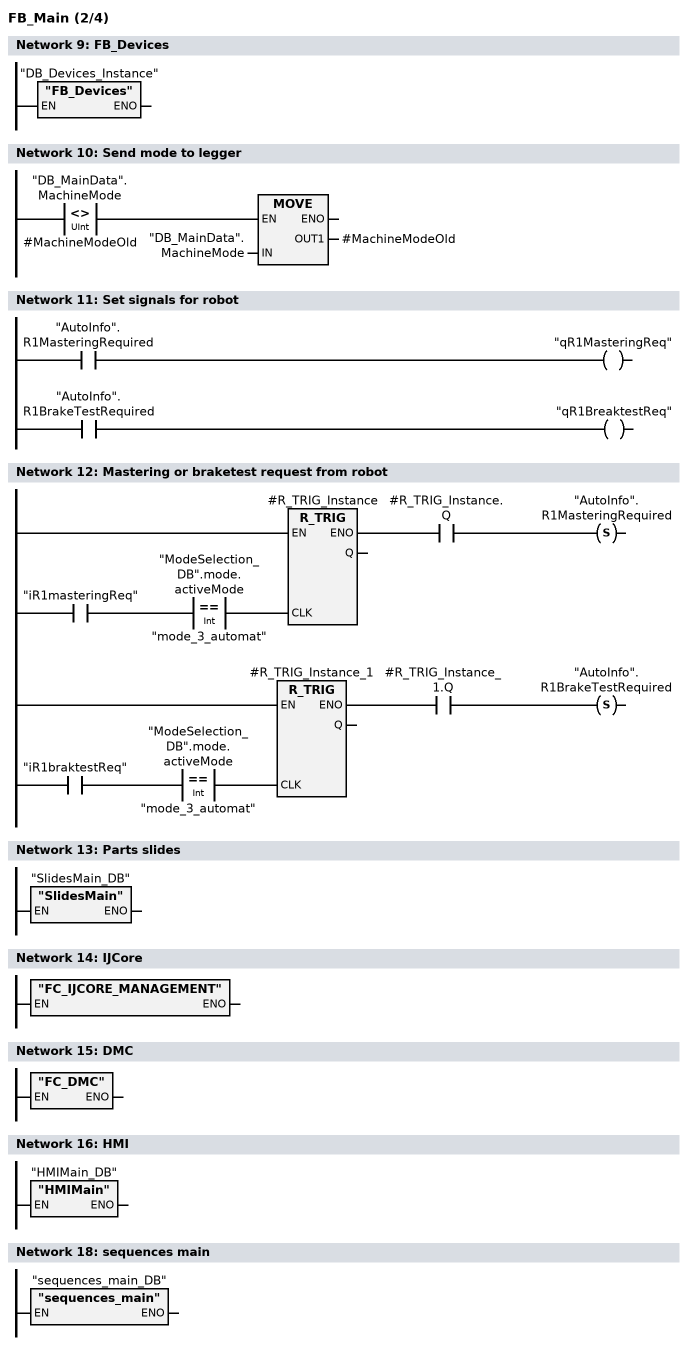
   RUNG wire#powerrail
      "DB_Devices_Instance"()
   END_RUNG
   // the same network as SCL:
   "DB_Devices_Instance"();   // "FB_Devices"
END_REGION

REGION Network 10: Send mode to legger
   RUNG wire#powerrail
      { S7_Templates := "SrcType := UInt" } NE_Contact(in1 := "DB_MainData".MachineMode, in2 := #MachineModeOld)
      Move(in := "DB_MainData".MachineMode, out1 => #MachineModeOld)
   END_RUNG
   // the same network as SCL:
   IF "DB_MainData".MachineMode <> #MachineModeOld THEN #MachineModeOld := "DB_MainData".MachineMode; END_IF;
END_REGION

REGION Network 11: Set signals for robot
   RUNG wire#powerrail
      Contact( "AutoInfo".R1MasteringRequired )
      Coil( "qR1MasteringReq" )
   END_RUNG
   RUNG wire#powerrail
      Contact( "AutoInfo".R1BrakeTestRequired )
      Coil( "qR1BreaktestReq" )
   END_RUNG
   // the same network as SCL:
   "qR1MasteringReq" := "AutoInfo".R1MasteringRequired;
   "qR1BreaktestReq" := "AutoInfo".R1BrakeTestRequired;
END_REGION

REGION Network 12: Mastering or braketest request from robot
   RUNG wire#powerrail
      #R_TRIG_Instance.R_TRIG(CLK := wire#w1, Q =>)
      Contact( #R_TRIG_Instance.Q )
      S_Coil( "AutoInfo".R1MasteringRequired )
   END_RUNG
   RUNG wire#powerrail
      Contact( "iR1masteringReq" )
      { S7_Templates := "SrcType := Int" } EQ_Contact(in1 := "ModeSelection_DB".mode.activeMode, in2 := "mode_3_automat")
   END_RUNG wire#w1
   RUNG wire#powerrail
      #R_TRIG_Instance_1.R_TRIG(CLK := wire#w2, Q =>)
      Contact( #R_TRIG_Instance_1.Q )
      S_Coil( "AutoInfo".R1BrakeTestRequired )
   END_RUNG
   RUNG wire#powerrail
      Contact( "iR1braktestReq" )
      { S7_Templates := "SrcType := Int" } EQ_Contact(in1 := "ModeSelection_DB".mode.activeMode, in2 := "mode_3_automat")
   END_RUNG wire#w2
   // the same network as SCL:
   #R_TRIG_Instance(CLK := "iR1masteringReq" AND ("ModeSelection_DB".mode.activeMode = "mode_3_automat"),   // R_TRIG
                    ENO => #_w1);
   IF #_w1 AND #R_TRIG_Instance.Q THEN "AutoInfo".R1MasteringRequired := TRUE; END_IF;
   #R_TRIG_Instance_1(CLK := "iR1braktestReq" AND ("ModeSelection_DB".mode.activeMode = "mode_3_automat"),   // R_TRIG
                      ENO => #_w2);
   IF #_w2 AND #R_TRIG_Instance_1.Q THEN "AutoInfo".R1BrakeTestRequired := TRUE; END_IF;
END_REGION

REGION Network 13: Parts slides
   RUNG wire#powerrail
      "SlidesMain_DB"()
   END_RUNG
   // the same network as SCL:
   "SlidesMain_DB"();   // "SlidesMain"
END_REGION

REGION Network 14: IJCore
   RUNG wire#powerrail
      "FC_IJCORE_MANAGEMENT"()
   END_RUNG
   // the same network as SCL:
   "FC_IJCORE_MANAGEMENT"();
END_REGION

REGION Network 15: DMC
   RUNG wire#powerrail
      "FC_DMC"()
   END_RUNG
   // the same network as SCL:
   "FC_DMC"();
END_REGION

REGION Network 16: HMI
   RUNG wire#powerrail
      "HMIMain_DB"()
   END_RUNG
   // the same network as SCL:
   "HMIMain_DB"();   // "HMIMain"
END_REGION

REGION Network 17 (SCL): mode selection
   "ModeSelection_DB"(iSafetyOKauto := "safety_signals"."4L+" AND NOT "SandBoxData".resetAuto,
                      iSafetyOKmanual := "safety_signals"."3L+",
                      iBasePosition := "sq_carousel_main_".base AND "sq_carousel_main_"."Base done".X AND
                      "sq_carousel_insertion_st1".base AND "sq_carousel_insertion_st1"."Base done".X AND
                      "sq_carousel_unloading_st2".base AND "sq_carousel_unloading_st2"."Base done".X AND
                      "sq_fitting_station_st3".base AND "sq_fitting_station_st3"."Base done".X AND
                      "sq_autoeject_DB".base AND "sq_autoeject_DB"."Base done".X AND
   //                   "sq_hanger_manipulator".base AND "sq_hanger_manipulator"."Base done".X AND
                      "sq_robot_".base AND "sq_robot_"."Base done".X,
                      iBaseInManualMode := TRUE,
                      OFF_SQ := FALSE,
                      INIT_SQ := TRUE,
                      SW_AUTO := TRUE);

   "ModeSelection_DB".mode.switch.auto := "iAuto" AND NOT "iManual";
   "ModeSelection_DB".mode.button.basic.request.button := "iBtnBasicPosition";
   "ModeSelection_DB".mode.button.auto.startRequest.button := "iBtnStartAuto";

   "DB_MainData".MachineMode := INT_TO_UINT("ModeSelection_DB".mode.activeMode);
   "SystemHMI".ManualMode := "ModeSelection_DB".mode.activeMode = "mode_1_manual";
   "SystemHMI".GoToBasicPosition := "ModeSelection_DB".mode.activeMode = "mode_2_base";
   "SystemHMI".AutomaticMode := "ModeSelection_DB".mode.activeMode = "mode_3_automat" OR "ModeSelection_DB".mode.activeMode = "mode_4_semiautomat";
   "SystemHMI".ModeChanged := "ModeSelection_DB".mode.modeChanged;

   "qBasicPosition" :=
   "ModeSelection_DB"."Base position reached".X OR
   "ModeSelection_DB".mode.activeMode = "mode_2_base" AND "Clock_5Hz" OR
   "ModeSelection_DB".mode.button.basic.request.visibility AND "Clock_1Hz";

   "qAuto" :=
   "ModeSelection_DB".mode.activeMode = "mode_3_automat" OR
   "ModeSelection_DB".mode.activeMode = "mode_4_semiautomat" OR
   "ModeSelection_DB".mode.button.auto.startRequest.visibility AND "Clock_1Hz";

   "qManual" := "ModeSelection_DB".mode.activeMode = "mode_1_manual";
END_REGION

REGION Network 18: sequences main
   RUNG wire#powerrail
      "sequences_main_DB"()
   END_RUNG
   // the same network as SCL:
   "sequences_main_DB"();   // "sequences_main"
END_REGION

REGION Network 19
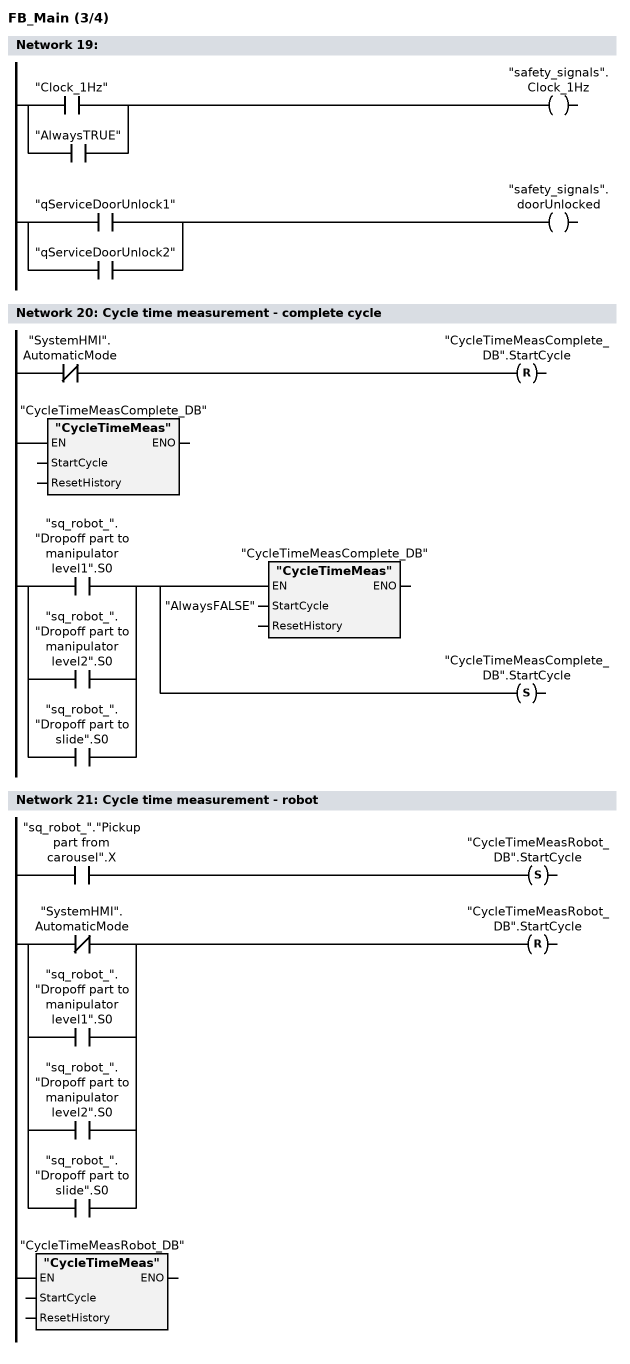
   RUNG wire#powerrail
      Contact( "Clock_1Hz" )
      wire#w1
      Coil( "safety_signals".Clock_1Hz )
   END_RUNG
   RUNG wire#powerrail
      Contact( "AlwaysTRUE" )
   END_RUNG wire#w1
   RUNG wire#powerrail
      Contact( "qServiceDoorUnlock1" )
      wire#w2
      Coil( "safety_signals".doorUnlocked )
   END_RUNG
   RUNG wire#powerrail
      Contact( "qServiceDoorUnlock2" )
   END_RUNG wire#w2
   // the same network as SCL:
   "safety_signals".Clock_1Hz := "Clock_1Hz" OR "AlwaysTRUE";
   "safety_signals".doorUnlocked := "qServiceDoorUnlock1" OR "qServiceDoorUnlock2";
END_REGION

REGION Network 20: Cycle time measurement - complete cycle
   RUNG wire#powerrail
      I_Contact( "SystemHMI".AutomaticMode )
      R_Coil( "CycleTimeMeasComplete_DB".StartCycle )
   END_RUNG
   RUNG wire#powerrail
      "CycleTimeMeasComplete_DB"(StartCycle :=, ResetHistory :=)
   END_RUNG
   RUNG wire#powerrail
      Contact( "sq_robot_"."Dropoff part to manipulator level1".S0 )
      wire#w1
      "CycleTimeMeasComplete_DB"(StartCycle := "AlwaysFALSE", ResetHistory :=)
   END_RUNG
   RUNG wire#powerrail
      Contact( "sq_robot_"."Dropoff part to manipulator level2".S0 )
   END_RUNG wire#w1
   RUNG wire#powerrail
      Contact( "sq_robot_"."Dropoff part to slide".S0 )
   END_RUNG wire#w1
   RUNG wire#w1
      S_Coil( "CycleTimeMeasComplete_DB".StartCycle )
   END_RUNG
   // the same network as SCL:
   IF NOT "SystemHMI".AutomaticMode THEN "CycleTimeMeasComplete_DB".StartCycle := FALSE; END_IF;
   "CycleTimeMeasComplete_DB"();   // "CycleTimeMeas"
   #_w1 := "sq_robot_"."Dropoff part to manipulator level1".S0 OR "sq_robot_"."Dropoff part to manipulator level2".S0 OR "sq_robot_"."Dropoff part to slide".S0;
   IF #_w1 THEN
       "CycleTimeMeasComplete_DB"(StartCycle := "AlwaysFALSE");   // "CycleTimeMeas"
       "CycleTimeMeasComplete_DB".StartCycle := TRUE;
   END_IF;
END_REGION

REGION Network 21: Cycle time measurement - robot
   RUNG wire#powerrail
      Contact( "sq_robot_"."Pickup part from carousel".X )
      S_Coil( "CycleTimeMeasRobot_DB".StartCycle )
   END_RUNG
   RUNG wire#powerrail
      I_Contact( "SystemHMI".AutomaticMode )
      wire#w1
      R_Coil( "CycleTimeMeasRobot_DB".StartCycle )
   END_RUNG
   RUNG wire#powerrail
      Contact( "sq_robot_"."Dropoff part to manipulator level1".S0 )
   END_RUNG wire#w1
   RUNG wire#powerrail
      Contact( "sq_robot_"."Dropoff part to manipulator level2".S0 )
   END_RUNG wire#w1
   RUNG wire#powerrail
      Contact( "sq_robot_"."Dropoff part to slide".S0 )
   END_RUNG wire#w1
   RUNG wire#powerrail
      "CycleTimeMeasRobot_DB"(StartCycle :=, ResetHistory :=)
   END_RUNG
   // the same network as SCL:
   IF "sq_robot_"."Pickup part from carousel".X THEN "CycleTimeMeasRobot_DB".StartCycle := TRUE; END_IF;
   IF NOT "SystemHMI".AutomaticMode OR "sq_robot_"."Dropoff part to manipulator level1".S0 OR "sq_robot_"."Dropoff part to manipulator level2".S0 OR "sq_robot_"."Dropoff part to slide".S0 THEN
       "CycleTimeMeasRobot_DB".StartCycle := FALSE;
   END_IF;
   "CycleTimeMeasRobot_DB"();   // "CycleTimeMeas"
END_REGION

REGION Network 22: Reset history
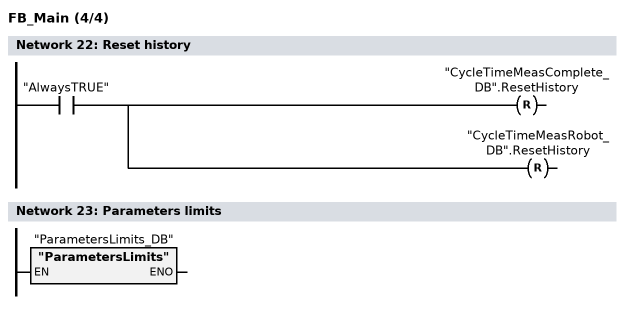
   RUNG wire#powerrail
      Contact( "AlwaysTRUE" )
      wire#w1
      R_Coil( "CycleTimeMeasComplete_DB".ResetHistory )
   END_RUNG
   RUNG wire#w1
      R_Coil( "CycleTimeMeasRobot_DB".ResetHistory )
   END_RUNG
   // the same network as SCL:
   IF "AlwaysTRUE" THEN
       "CycleTimeMeasComplete_DB".ResetHistory := FALSE;
       "CycleTimeMeasRobot_DB".ResetHistory := FALSE;
   END_IF;
END_REGION

REGION Network 23: Parameters limits
   RUNG wire#powerrail
      "ParametersLimits_DB"()
   END_RUNG
   // the same network as SCL:
   "ParametersLimits_DB"();   // "ParametersLimits"
END_REGION
END_FUNCTION_BLOCK

FUNCTION_BLOCK "FB_Eks"   // FB5050, LAD
{ S7_Optimized_Access := 'TRUE' }
VERSION : 0.1
// stored: AutoNumber false, IsIECCheckEnabled false, IsRetainMemResEnabled false, MemoryReserve 100, SetENOAutomatically false, UDAEnableTagReadback false
   VAR_INPUT
      iScreenNumberEqual : Bool;
      iOpSwitchManualMode : Bool;
      iGenerateTimeoutError : Bool;
      iPermanentAccess : Bool;
      iBlinker : Bool;
   END_VAR
   VAR_OUTPUT
      qManualModeActive : Bool;
      qOpManualModeLamp : Bool;
      qeKeyTimeout : Bool;
   END_VAR
   VAR DB_SPECIFIC
      Status : Struct
         Key : Struct
            Inserted : Bool;
            Found : Bool;
            Valid : Bool;
            ActualKeyStatus : Int;   // 0= Not inserted, ??= GAP leader, ??= Maintenance, ??= Engineer, 100= Not registered
            LastKeyStatus : Int;   // 0= Not used, ??= GAP leader, ??= Maintenance, ??= Engineer, 100= Not registered
         END_STRUCT;
         Global : Struct
            GapLeader : Bool;
            Maintenance : Bool;
            Engineer : Bool;
            MaintenanceOrEngineer : Bool;
            AnyValidKey : Bool;
         END_STRUCT;
         ManualMode : Struct
            GapLeader : Bool;
            Maintenance : Bool;
            Engineer : Bool;
            MaintenanceOrEngineer : Bool;
            AnyValidKey : Bool;
         END_STRUCT;
      END_STRUCT;
   END_VAR
   VAR
      Database : Struct
         Status : Struct
            ActualAndLastKeyEqual { ExternalAccessible := 'False'; ExternalVisible := 'False'; ExternalWritable := 'False'} : Bool;
            LastKeyIsEmpty : Bool;
            LastKeyEmployeeIDIsEmpty : Bool;
            LastKeyFound { ExternalAccessible := 'False'; ExternalVisible := 'False'; ExternalWritable := 'False'} : Bool;
            LastKeyIndex { ExternalAccessible := 'False'; ExternalVisible := 'False'; ExternalWritable := 'False'} : Int;
            FreePlaceFound { ExternalAccessible := 'False'; ExternalVisible := 'False'; ExternalWritable := 'False'} : Bool;
            FreePlaceIndex { ExternalAccessible := 'False'; ExternalVisible := 'False'; ExternalWritable := 'False'} : Int;
            NumberOfKeys : Int;
            NumberOfStoredKeys : Int;
            StoredKeysReachedMaximum : Bool;
            NumberOfEngineerKeys : Int;
            NumberOfStoredEngineerKeys : Int;
            StoredEngineerKeysReachedMaximum : Bool;
         END_STRUCT;
         ListNumber : Int;
         ListNumberLast : Int;
      END_STRUCT;
   END_VAR
   VAR DB_SPECIFIC
      KeyManage : Struct
         CanBeAdd : Bool;
         Add : Bool;
         CanBeRemoved : Bool;
         Remove : Bool;
         CanBeUsed : Bool;
         Use : Int;
         CanBeSearched : Bool;
         Search : Bool;
         Searching : Bool;
         SearchedRow : Int;
         SearchedRowHMI : Int;
      END_STRUCT;
   END_VAR
   VAR RETAIN
      KeyTimeout : Time := T#2H_46M_39S;
   END_VAR
   VAR
      KeyInsertedInReader { S7_SetPoint := 'True'} : R_TRIG;
      KeyRemovedFromReader { S7_SetPoint := 'True'} : F_TRIG;
   END_VAR
   VAR DB_SPECIFIC
      TONs : Struct
         tDelayTimeoutError { S7_SetPoint := 'True'} : TON_TIME;
      END_STRUCT;
   END_VAR
   VAR_TEMP
      i : Int;
      stored_keys : Int;
      stored_engineer_keys : Int;
   END_VAR
   VAR_TEMP   // added for the SCL form of the ladder/FBD networks
      _w1 : Bool;
   END_VAR
BEGIN

REGION Network 1 (SCL): Inserted key
   //Key is inserted in reader
   #KeyInsertedInReader(CLK := "iEksKeyInserted");

   IF #KeyInsertedInReader.Q THEN
       "DB_EksData".LoadedData := "DB_EksData".EmptyKey;
       "DB_EksData".ActualKey := "DB_EksData".EmptyKey;
       #Status.Key.Inserted := TRUE;

       //Load level
       "DB_EksData".LoadedData.Level := "iEksLevel";

       //Load employee ID 
       "DB_EksData".LoadedData.EmployeeID[1] := "iEksEmployeeID_1";
       "DB_EksData".LoadedData.EmployeeID[2] := "iEksEmployeeID_2";
       "DB_EksData".LoadedData.EmployeeID[3] := "iEksEmployeeID_3";
       "DB_EksData".LoadedData.EmployeeID[4] := "iEksEmployeeID_4";

       //Adjust employee ID to be sure, that comparing with empty data will be coorect
       FOR #i := 1 TO 4 DO
           IF "DB_EksData".LoadedData.EmployeeID[#i] = '$00' THEN
               "DB_EksData".LoadedData.EmployeeID[#i] := ' ';
           END_IF;
       END_FOR;

       //Load key ID
       "FC_ByteToCharacters"(iByte := "iEksKeyID_1",
                             qChar1 => "DB_EksData".LoadedData.KeyID[1],
                             qChar2 => "DB_EksData".LoadedData.KeyID[2]);
       "FC_ByteToCharacters"(iByte := "iEksKeyID_2",
                             qChar1 => "DB_EksData".LoadedData.KeyID[3],
                             qChar2 => "DB_EksData".LoadedData.KeyID[4]);
       "FC_ByteToCharacters"(iByte := "iEksKeyID_3",
                             qChar1 => "DB_EksData".LoadedData.KeyID[5],
                             qChar2 => "DB_EksData".LoadedData.KeyID[6]);
       "FC_ByteToCharacters"(iByte := "iEksKeyID_4",
                             qChar1 => "DB_EksData".LoadedData.KeyID[7],
                             qChar2 => "DB_EksData".LoadedData.KeyID[8]);
       "FC_ByteToCharacters"(iByte := "iEksKeyID_5",
                             qChar1 => "DB_EksData".LoadedData.KeyID[9],
                             qChar2 => "DB_EksData".LoadedData.KeyID[10]);
       "FC_ByteToCharacters"(iByte := "iEksKeyID_6",
                             qChar1 => "DB_EksData".LoadedData.KeyID[11],
                             qChar2 => "DB_EksData".LoadedData.KeyID[12]);
       "FC_ByteToCharacters"(iByte := "iEksKeyID_7",
                             qChar1 => "DB_EksData".LoadedData.KeyID[13],
                             qChar2 => "DB_EksData".LoadedData.KeyID[14]);
       "FC_ByteToCharacters"(iByte := "iEksKeyID_8",
                             qChar1 => "DB_EksData".LoadedData.KeyID[15],
                             qChar2 => "DB_EksData".LoadedData.KeyID[16]);

       //Search inserted key in database
       FOR #i := 1 TO "EksNumberOfKeys" DO
           IF "DB_EksData".LoadedData.KeyID = "DB_EksList".Key[#i].KeyID THEN
               "DB_EksData".ActualKey := "DB_EksList".Key[#i];
               #Status.Key.Found := TRUE;
               IF "DB_EksList".Key[#i].Level = "EksGapLeaderLevel" OR
                   "DB_EksList".Key[#i].Level = "EksMaintenanceLevel" OR
                   "DB_EksList".Key[#i].Level = "EksEngineerLevel" THEN
                   #Status.Key.Valid := TRUE;
               END_IF;
               EXIT;
           END_IF;
       END_FOR;
       IF NOT #Status.Key.Found THEN
           "DB_EksData".ActualKey := "DB_EksData".LoadedData;
       END_IF;
   END_IF;

   //Key is removed from reader
   #KeyRemovedFromReader(CLK:="iEksKeyInserted");

   IF #KeyRemovedFromReader.Q THEN
       "DB_EksData".LastKey := "DB_EksData".ActualKey;
       "DB_EksData".ActualKey := "DB_EksData".EmptyKey;
   END_IF;

   //Manage data when key is not in reader or timeout error
   IF NOT "iEksKeyInserted" OR #qeKeyTimeout THEN
       #Status.Key.Inserted := FALSE;
       #Status.Key.Found := FALSE;
       #Status.Key.Valid := FALSE;
       #Status.Key.ActualKeyStatus := 0;
       "DB_EksData".ActualKey := "DB_EksData".EmptyKey;
   END_IF;

   //Reset timeout error
   IF NOT "iEksKeyInserted" THEN
       #qeKeyTimeout := FALSE;
   END_IF;
END_REGION

REGION Network 2: Set key status
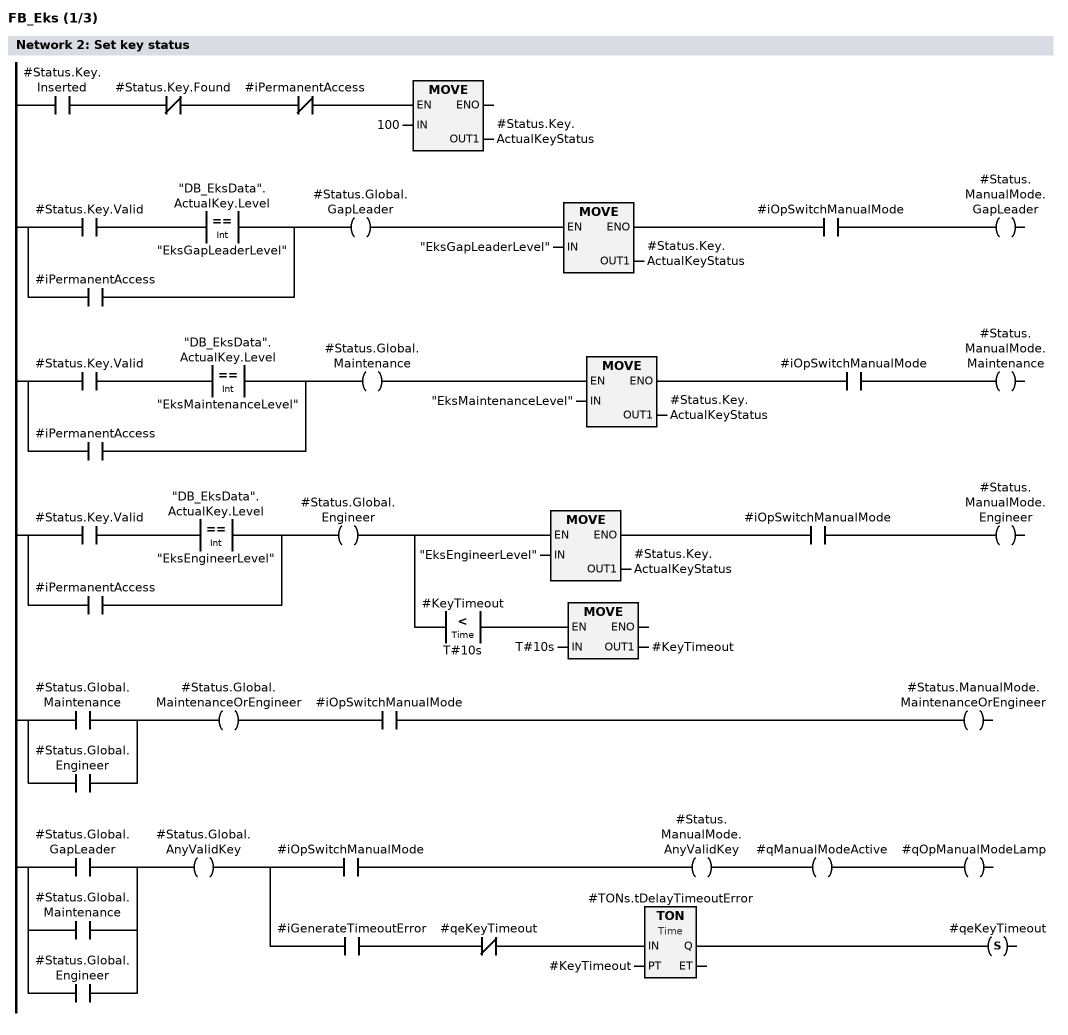
   RUNG wire#powerrail
      Contact( #Status.Key.Inserted )
      I_Contact( #Status.Key.Found )
      I_Contact( #iPermanentAccess )
      Move(in := 100, out1 => #Status.Key.ActualKeyStatus)
   END_RUNG
   RUNG wire#powerrail
      Contact( #Status.Key.Valid )
      { S7_Templates := "SrcType := Int" } EQ_Contact(in1 := "DB_EksData".ActualKey.Level, in2 := "EksGapLeaderLevel")
      wire#w1
      Coil( #Status.Global.GapLeader )
      Move(in := "EksGapLeaderLevel", out1 => #Status.Key.ActualKeyStatus)
      Contact( #iOpSwitchManualMode )
      Coil( #Status.ManualMode.GapLeader )
   END_RUNG
   RUNG wire#powerrail
      Contact( #iPermanentAccess )
   END_RUNG wire#w1
   RUNG wire#powerrail
      Contact( #Status.Key.Valid )
      { S7_Templates := "SrcType := Int" } EQ_Contact(in1 := "DB_EksData".ActualKey.Level, in2 := "EksMaintenanceLevel")
      wire#w2
      Coil( #Status.Global.Maintenance )
      Move(in := "EksMaintenanceLevel", out1 => #Status.Key.ActualKeyStatus)
      Contact( #iOpSwitchManualMode )
      Coil( #Status.ManualMode.Maintenance )
   END_RUNG
   RUNG wire#powerrail
      Contact( #iPermanentAccess )
   END_RUNG wire#w2
   RUNG wire#powerrail
      Contact( #Status.Key.Valid )
      { S7_Templates := "SrcType := Int" } EQ_Contact(in1 := "DB_EksData".ActualKey.Level, in2 := "EksEngineerLevel")
      wire#w3
      Coil( #Status.Global.Engineer )
      wire#w4
      Move(in := "EksEngineerLevel", out1 => #Status.Key.ActualKeyStatus)
      Contact( #iOpSwitchManualMode )
      Coil( #Status.ManualMode.Engineer )
   END_RUNG
   RUNG wire#powerrail
      Contact( #iPermanentAccess )
   END_RUNG wire#w3
   RUNG wire#w4
      { S7_Templates := "SrcType := Time" } LT_Contact(in1 := #KeyTimeout, in2 := T#10s)
      Move(in := T#10s, out1 => #KeyTimeout)
   END_RUNG
   RUNG wire#powerrail
      Contact( #Status.Global.Maintenance )
      wire#w5
      Coil( #Status.Global.MaintenanceOrEngineer )
      Contact( #iOpSwitchManualMode )
      Coil( #Status.ManualMode.MaintenanceOrEngineer )
   END_RUNG
   RUNG wire#powerrail
      Contact( #Status.Global.Engineer )
   END_RUNG wire#w5
   RUNG wire#powerrail
      Contact( #Status.Global.GapLeader )
      wire#w6
      Coil( #Status.Global.AnyValidKey )
      wire#w7
      Contact( #iOpSwitchManualMode )
      Coil( #Status.ManualMode.AnyValidKey )
      Coil( #qManualModeActive )
      Coil( #qOpManualModeLamp )
   END_RUNG
   RUNG wire#powerrail
      Contact( #Status.Global.Maintenance )
   END_RUNG wire#w6
   RUNG wire#powerrail
      Contact( #Status.Global.Engineer )
   END_RUNG wire#w6
   RUNG wire#w7
      Contact( #iGenerateTimeoutError )
      I_Contact( #qeKeyTimeout )
      { S7_Templates := "time_type := Time" } #TONs.tDelayTimeoutError.TON(pt := #KeyTimeout, et =>)
      S_Coil( #qeKeyTimeout )
   END_RUNG
   // the same network as SCL:
   IF #Status.Key.Inserted AND NOT #Status.Key.Found AND NOT #iPermanentAccess THEN
       #Status.Key.ActualKeyStatus := 100;
   END_IF;
   #Status.Global.GapLeader := (#Status.Key.Valid AND ("DB_EksData".ActualKey.Level = "EksGapLeaderLevel")) OR #iPermanentAccess;
   IF #Status.Global.GapLeader THEN #Status.Key.ActualKeyStatus := "EksGapLeaderLevel"; END_IF;
   #Status.ManualMode.GapLeader := #Status.Global.GapLeader AND #iOpSwitchManualMode;
   #Status.Global.Maintenance := (#Status.Key.Valid AND ("DB_EksData".ActualKey.Level = "EksMaintenanceLevel")) OR #iPermanentAccess;
   IF #Status.Global.Maintenance THEN #Status.Key.ActualKeyStatus := "EksMaintenanceLevel"; END_IF;
   #Status.ManualMode.Maintenance := #Status.Global.Maintenance AND #iOpSwitchManualMode;
   #Status.Global.Engineer := (#Status.Key.Valid AND ("DB_EksData".ActualKey.Level = "EksEngineerLevel")) OR #iPermanentAccess;
   IF #Status.Global.Engineer THEN #Status.Key.ActualKeyStatus := "EksEngineerLevel"; END_IF;
   #Status.ManualMode.Engineer := #Status.Global.Engineer AND #iOpSwitchManualMode;
   IF #Status.Global.Engineer AND (#KeyTimeout < T#10s) THEN #KeyTimeout := T#10s; END_IF;
   #Status.Global.MaintenanceOrEngineer := #Status.Global.Maintenance OR #Status.Global.Engineer;
   #Status.ManualMode.MaintenanceOrEngineer := #Status.Global.MaintenanceOrEngineer AND #iOpSwitchManualMode;
   #Status.Global.AnyValidKey := #Status.Global.GapLeader OR #Status.Global.Maintenance OR #Status.Global.Engineer;
   #Status.ManualMode.AnyValidKey := #Status.Global.AnyValidKey AND #iOpSwitchManualMode;
   #qManualModeActive := #Status.ManualMode.AnyValidKey;
   #qOpManualModeLamp := #Status.ManualMode.AnyValidKey;
   #TONs.tDelayTimeoutError.TON(IN := #Status.Global.AnyValidKey AND #iGenerateTimeoutError AND NOT #qeKeyTimeout,
                           PT := #KeyTimeout);
   IF #TONs.tDelayTimeoutError.Q THEN #qeKeyTimeout := TRUE; END_IF;
END_REGION

REGION Network 3 (SCL): Database status
   //Database status
   IF #iScreenNumberEqual THEN

       //Reset database status
       #Database.Status.ActualAndLastKeyEqual := FALSE;
       #Database.Status.LastKeyIsEmpty := FALSE;
       #Database.Status.LastKeyEmployeeIDIsEmpty := FALSE;
       #Database.Status.LastKeyFound := FALSE;
       #Database.Status.LastKeyIndex := 0;
       #Database.Status.FreePlaceFound := FALSE;
       #Database.Status.FreePlaceIndex := 0;
       #stored_keys := 0;
       #stored_engineer_keys := 0;

       //Compare actual and last inserted key
       IF #Status.Key.Inserted AND "DB_EksData".ActualKey.KeyID = "DB_EksData".LastKey.KeyID THEN
           //"DB_EksData".ActualKey.EmployeeID <> "DB_EksData".EmptyKey.EmployeeID THEN
           #Database.Status.ActualAndLastKeyEqual := TRUE;
       END_IF;

       //Last key is empty
       IF "DB_EksData".LastKey = "DB_EksData".EmptyKey THEN
           #Database.Status.LastKeyIsEmpty := TRUE;
       END_IF;

       //Last key employee ID is empty
       IF "DB_EksData".LastKey.EmployeeID = "DB_EksData".EmptyKey.EmployeeID THEN
           #Database.Status.LastKeyEmployeeIDIsEmpty := TRUE;
       END_IF;

       //Search database
       FOR #i := 1 TO "EksNumberOfKeys" DO

           //Search last key in database
           IF NOT #Database.Status.LastKeyFound AND
               "DB_EksData".LastKey.KeyID = "DB_EksList".Key[#i].KeyID THEN
               #Database.Status.LastKeyFound := TRUE;
               #Database.Status.LastKeyIndex := #i;
               #Status.Key.LastKeyStatus := "DB_EksData".LastKey.Level;
           END_IF;

           //Search free place in database            
           IF NOT #Database.Status.FreePlaceFound AND "DB_EksList".Key[#i] = "DB_EksData".EmptyKey THEN
               #Database.Status.FreePlaceFound := TRUE;
               #Database.Status.FreePlaceIndex := #i;
           END_IF;

           //Count stored keys
           IF "DB_EksList".Key[#i] <> "DB_EksData".EmptyKey THEN
               #stored_keys := #stored_keys + 1;

               IF "DB_EksList".Key[#i].Level = "EksEngineerLevel" THEN
                   #stored_engineer_keys := #stored_engineer_keys + 1;
               END_IF;

           END_IF;

       END_FOR;

       //Last key is not used
       IF #Database.Status.LastKeyIsEmpty THEN
           #Status.Key.LastKeyStatus := 0;
       END_IF;

       //Last key is not registered
       IF NOT #Database.Status.LastKeyIsEmpty AND NOT #Database.Status.LastKeyFound THEN
           #Status.Key.LastKeyStatus := 100;
       END_IF;

       //Check number of stored keys
       #Database.Status.NumberOfStoredKeys := #stored_keys;
       IF #Database.Status.NumberOfStoredKeys >= "EksNumberOfKeys" THEN
           #Database.Status.StoredKeysReachedMaximum := TRUE;
       ELSE
           #Database.Status.StoredKeysReachedMaximum := FALSE;
       END_IF;

       //Check number of stored engineer keys
       #Database.Status.NumberOfStoredEngineerKeys := #stored_engineer_keys;
       IF #Database.Status.NumberOfStoredEngineerKeys >= "EksNumberOfEngineerKeys" THEN
           #Database.Status.StoredEngineerKeysReachedMaximum := TRUE;
       ELSE
           #Database.Status.StoredEngineerKeysReachedMaximum := FALSE;
       END_IF;

   END_IF;
END_REGION

REGION Network 4: Add key
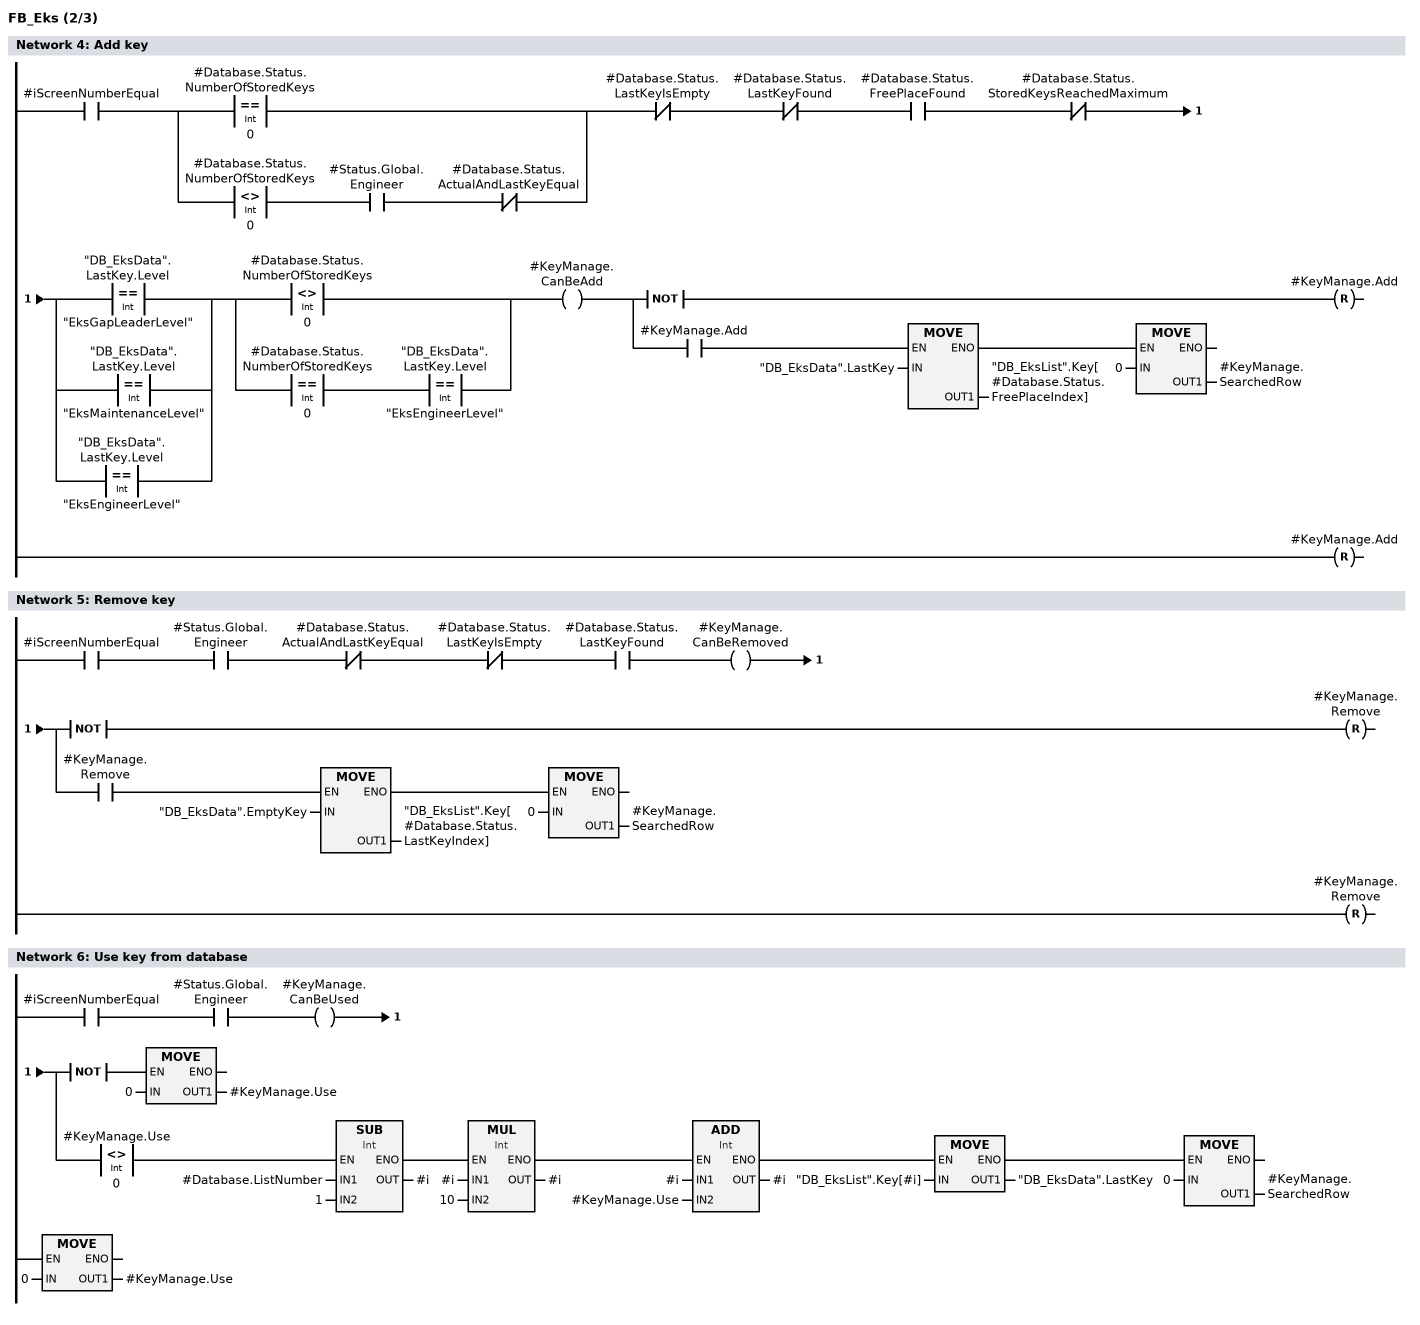
   RUNG wire#powerrail
      Contact( #iScreenNumberEqual )
      wire#w1
      { S7_Templates := "SrcType := Int" } EQ_Contact(in1 := #Database.Status.NumberOfStoredKeys, in2 := 0)
      wire#w2
      I_Contact( #Database.Status.LastKeyIsEmpty )
      I_Contact( #Database.Status.LastKeyFound )
      Contact( #Database.Status.FreePlaceFound )
      I_Contact( #Database.Status.StoredKeysReachedMaximum )
      wire#w3
      { S7_Templates := "SrcType := Int" } EQ_Contact(in1 := "DB_EksData".LastKey.Level, in2 := "EksGapLeaderLevel")
      wire#w4
      { S7_Templates := "SrcType := Int" } NE_Contact(in1 := #Database.Status.NumberOfStoredKeys, in2 := 0)
      wire#w5
      Coil( #KeyManage.CanBeAdd )
      wire#w6
      Not()
      R_Coil( #KeyManage.Add )
   END_RUNG
   RUNG wire#w1
      { S7_Templates := "SrcType := Int" } NE_Contact(in1 := #Database.Status.NumberOfStoredKeys, in2 := 0)
      Contact( #Status.Global.Engineer )
      I_Contact( #Database.Status.ActualAndLastKeyEqual )
   END_RUNG wire#w2
   RUNG wire#w3
      { S7_Templates := "SrcType := Int" } EQ_Contact(in1 := "DB_EksData".LastKey.Level, in2 := "EksMaintenanceLevel")
   END_RUNG wire#w4
   RUNG wire#w3
      { S7_Templates := "SrcType := Int" } EQ_Contact(in1 := "DB_EksData".LastKey.Level, in2 := "EksEngineerLevel")
   END_RUNG wire#w4
   RUNG wire#w4
      { S7_Templates := "SrcType := Int" } EQ_Contact(in1 := #Database.Status.NumberOfStoredKeys, in2 := 0)
      { S7_Templates := "SrcType := Int" } EQ_Contact(in1 := "DB_EksData".LastKey.Level, in2 := "EksEngineerLevel")
   END_RUNG wire#w5
   RUNG wire#w6
      Contact( #KeyManage.Add )
      Move(in := "DB_EksData".LastKey, out1 => "DB_EksList".Key[#Database.Status.FreePlaceIndex])
      Move(in := 0, out1 => #KeyManage.SearchedRow)
   END_RUNG
   RUNG wire#powerrail
      R_Coil( #KeyManage.Add )
   END_RUNG
   // the same network as SCL:
   #KeyManage.CanBeAdd := #iScreenNumberEqual AND ((#Database.Status.NumberOfStoredKeys = 0) OR ((#Database.Status.NumberOfStoredKeys <> 0) AND #Status.Global.Engineer AND NOT #Database.Status.ActualAndLastKeyEqual)) AND NOT #Database.Status.LastKeyIsEmpty AND NOT #Database.Status.LastKeyFound AND #Database.Status.FreePlaceFound AND NOT #Database.Status.StoredKeysReachedMaximum AND (("DB_EksData".LastKey.Level = "EksGapLeaderLevel") OR ("DB_EksData".LastKey.Level = "EksMaintenanceLevel") OR ("DB_EksData".LastKey.Level = "EksEngineerLevel")) AND ((#Database.Status.NumberOfStoredKeys <> 0) OR ((#Database.Status.NumberOfStoredKeys = 0) AND ("DB_EksData".LastKey.Level = "EksEngineerLevel")));
   IF NOT #KeyManage.CanBeAdd THEN #KeyManage.Add := FALSE; END_IF;
   IF #KeyManage.CanBeAdd AND #KeyManage.Add THEN
       "DB_EksList".Key[#Database.Status.FreePlaceIndex] := "DB_EksData".LastKey;
       #KeyManage.SearchedRow := 0;
   END_IF;
   #KeyManage.Add := FALSE;
END_REGION

REGION Network 5: Remove key
   RUNG wire#powerrail
      Contact( #iScreenNumberEqual )
      Contact( #Status.Global.Engineer )
      I_Contact( #Database.Status.ActualAndLastKeyEqual )
      I_Contact( #Database.Status.LastKeyIsEmpty )
      Contact( #Database.Status.LastKeyFound )
      Coil( #KeyManage.CanBeRemoved )
      wire#w1
      Not()
      R_Coil( #KeyManage.Remove )
   END_RUNG
   RUNG wire#w1
      Contact( #KeyManage.Remove )
      Move(in := "DB_EksData".EmptyKey, out1 => "DB_EksList".Key[#Database.Status.LastKeyIndex])
      Move(in := 0, out1 => #KeyManage.SearchedRow)
   END_RUNG
   RUNG wire#powerrail
      R_Coil( #KeyManage.Remove )
   END_RUNG
   // the same network as SCL:
   #KeyManage.CanBeRemoved := #iScreenNumberEqual AND #Status.Global.Engineer AND NOT #Database.Status.ActualAndLastKeyEqual AND NOT #Database.Status.LastKeyIsEmpty AND #Database.Status.LastKeyFound;
   IF NOT #KeyManage.CanBeRemoved THEN #KeyManage.Remove := FALSE; END_IF;
   IF #KeyManage.CanBeRemoved AND #KeyManage.Remove THEN
       "DB_EksList".Key[#Database.Status.LastKeyIndex] := "DB_EksData".EmptyKey;
       #KeyManage.SearchedRow := 0;
   END_IF;
   #KeyManage.Remove := FALSE;
END_REGION

REGION Network 6: Use key from database
   RUNG wire#powerrail
      Contact( #iScreenNumberEqual )
      Contact( #Status.Global.Engineer )
      Coil( #KeyManage.CanBeUsed )
      wire#w1
      Not()
      Move(in := 0, out1 => #KeyManage.Use)
   END_RUNG
   RUNG wire#w1
      { S7_Templates := "SrcType := Int" } NE_Contact(in1 := #KeyManage.Use, in2 := 0)
      { S7_Templates := "SrcType := Int" } Sub(in1 := #Database.ListNumber, in2 := 1, out => #i)
      { S7_Templates := "SrcType := Int" } Mul(in1 := #i, in2 := 10, out => #i)
      { S7_Templates := "SrcType := Int" } Add(in1 := #i, in2 := #KeyManage.Use, out => #i)
      Move(in := "DB_EksList".Key[#i], out1 => "DB_EksData".LastKey)
      Move(in := 0, out1 => #KeyManage.SearchedRow)
   END_RUNG
   RUNG wire#powerrail
      Move(in := 0, out1 => #KeyManage.Use)
   END_RUNG
   // the same network as SCL:
   #KeyManage.CanBeUsed := #iScreenNumberEqual AND #Status.Global.Engineer;
   IF NOT #KeyManage.CanBeUsed THEN #KeyManage.Use := 0; END_IF;
   IF #KeyManage.CanBeUsed AND (#KeyManage.Use <> 0) THEN
       #i := #Database.ListNumber - 1;
       #i := #i * 10;
       #i := #i + #KeyManage.Use;
       "DB_EksData".LastKey := "DB_EksList".Key[#i];
       #KeyManage.SearchedRow := 0;
   END_IF;
   #KeyManage.Use := 0;
END_REGION

REGION Network 7: Search last inserted key
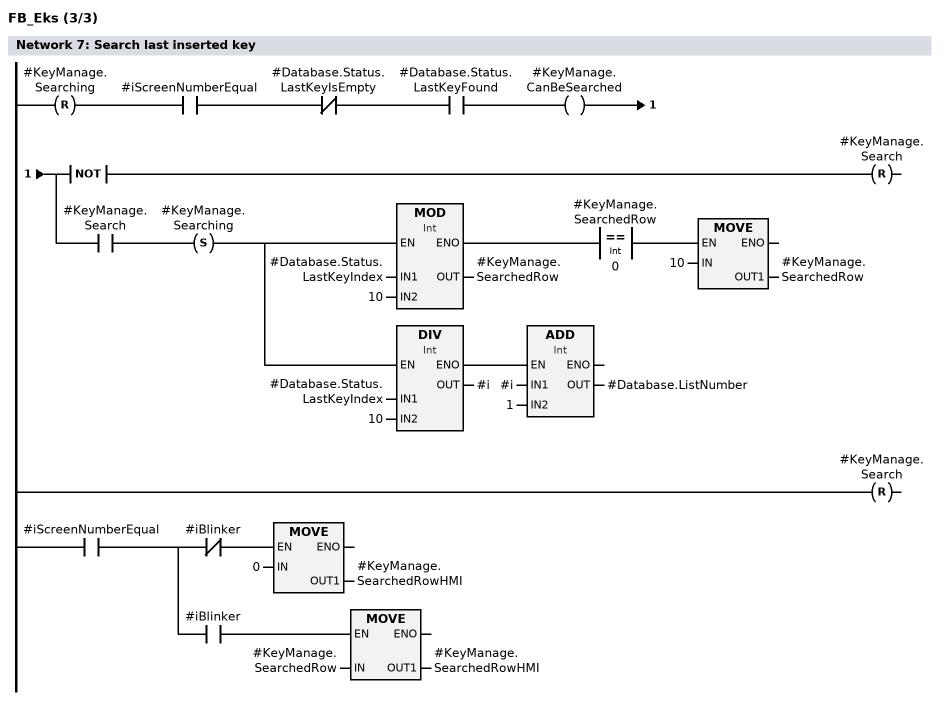
   RUNG wire#powerrail
      R_Coil( #KeyManage.Searching )
      Contact( #iScreenNumberEqual )
      I_Contact( #Database.Status.LastKeyIsEmpty )
      Contact( #Database.Status.LastKeyFound )
      Coil( #KeyManage.CanBeSearched )
      wire#w1
      Not()
      R_Coil( #KeyManage.Search )
   END_RUNG
   RUNG wire#w1
      Contact( #KeyManage.Search )
      S_Coil( #KeyManage.Searching )
      wire#w2
      { S7_Templates := "SrcType := Int" } Mod(in1 := #Database.Status.LastKeyIndex, in2 := 10, out => #KeyManage.SearchedRow)
      { S7_Templates := "SrcType := Int" } EQ_Contact(in1 := #KeyManage.SearchedRow, in2 := 0)
      Move(in := 10, out1 => #KeyManage.SearchedRow)
   END_RUNG
   RUNG wire#w2
      { S7_Templates := "SrcType := Int" } Div(in1 := #Database.Status.LastKeyIndex, in2 := 10, out => #i)
      { S7_Templates := "SrcType := Int" } Add(in1 := #i, in2 := 1, out => #Database.ListNumber)
   END_RUNG
   RUNG wire#powerrail
      R_Coil( #KeyManage.Search )
   END_RUNG
   RUNG wire#powerrail
      Contact( #iScreenNumberEqual )
      wire#w3
      I_Contact( #iBlinker )
      Move(in := 0, out1 => #KeyManage.SearchedRowHMI)
   END_RUNG
   RUNG wire#w3
      Contact( #iBlinker )
      Move(in := #KeyManage.SearchedRow, out1 => #KeyManage.SearchedRowHMI)
   END_RUNG
   // the same network as SCL:
   #KeyManage.Searching := FALSE;
   #KeyManage.CanBeSearched := #iScreenNumberEqual AND NOT #Database.Status.LastKeyIsEmpty AND #Database.Status.LastKeyFound;
   IF NOT #KeyManage.CanBeSearched THEN #KeyManage.Search := FALSE; END_IF;
   #_w1 := #KeyManage.CanBeSearched AND #KeyManage.Search;
   IF #_w1 THEN
       #KeyManage.Searching := TRUE;
       #KeyManage.SearchedRow := #Database.Status.LastKeyIndex MOD 10;
   END_IF;
   IF #_w1 AND (#KeyManage.SearchedRow = 0) THEN #KeyManage.SearchedRow := 10; END_IF;
   IF #_w1 THEN
       #i := #Database.Status.LastKeyIndex / 10;
       #Database.ListNumber := #i + 1;
   END_IF;
   #KeyManage.Search := FALSE;
   IF #iScreenNumberEqual AND NOT #iBlinker THEN #KeyManage.SearchedRowHMI := 0; END_IF;
   IF #iScreenNumberEqual AND #iBlinker THEN #KeyManage.SearchedRowHMI := #KeyManage.SearchedRow; END_IF;
END_REGION

REGION Network 8 (SCL): Key listing
   //List number limits
   IF #Database.ListNumber < 1 THEN
       #Database.ListNumber := 1;
   END_IF;

   #i := "EksNumberOfKeys" / 10;
   IF #Database.ListNumber > #i THEN
       #Database.ListNumber := #i;
   END_IF;

   //Keys limit
   #Database.Status.NumberOfKeys := "EksNumberOfKeys";
   #Database.Status.NumberOfEngineerKeys := "EksNumberOfEngineerKeys";

   //Reset searched row
   IF NOT #iScreenNumberEqual THEN
       #KeyManage.SearchedRow := 0;
   END_IF;

   IF #Database.ListNumberLast <> #Database.ListNumber THEN
       #Database.ListNumberLast := #Database.ListNumber;

       IF NOT #KeyManage.Searching THEN
           #KeyManage.SearchedRow := 0;
       END_IF;

   END_IF;

   //Key listing
   IF #iScreenNumberEqual THEN
       #i := (#Database.ListNumber - 1) * 10;
       "DB_EksData".KeyListHMI[1] := "DB_EksList".Key[#i + 1];
       "DB_EksData".KeyListHMI[2] := "DB_EksList".Key[#i + 2];
       "DB_EksData".KeyListHMI[3] := "DB_EksList".Key[#i + 3];
       "DB_EksData".KeyListHMI[4] := "DB_EksList".Key[#i + 4];
       "DB_EksData".KeyListHMI[5] := "DB_EksList".Key[#i + 5];
       "DB_EksData".KeyListHMI[6] := "DB_EksList".Key[#i + 6];
       "DB_EksData".KeyListHMI[7] := "DB_EksList".Key[#i + 7];
       "DB_EksData".KeyListHMI[8] := "DB_EksList".Key[#i + 8];
       "DB_EksData".KeyListHMI[9] := "DB_EksList".Key[#i + 9];
       "DB_EksData".KeyListHMI[10] := "DB_EksList".Key[#i + 10];
   END_IF;
END_REGION
END_FUNCTION_BLOCK

FUNCTION_BLOCK "FB_DateTimeAndShifts"   // FB5010, LAD
{ S7_Optimized_Access := 'TRUE' }
VERSION : 0.1
// stored: AutoNumber false, IsIECCheckEnabled false, IsRetainMemResEnabled false, MemoryReserve 100, SetENOAutomatically false, UDAEnableTagReadback false
   VAR_INPUT
      iSettingsSecurity : Bool;
   END_VAR
   VAR
      Edges : Struct
         Shift1Started : Bool;
         Shift2Started : Bool;
         Shift3Started : Bool;
      END_STRUCT;
   END_VAR
   VAR RETAIN
      Settings : Struct
         Actual { S7_SetPoint := 'True'} : "UDT_DateTimeAndShiftsSettings";
         Last { S7_SetPoint := 'True'} : "UDT_DateTimeAndShiftsSettings";
         Status : Struct
            SettingsCanBeChanged : Bool;   // 0= No
         END_STRUCT;
         Commands : Struct
            DateAndTimeUse : Bool;
            DateAndTimeSet : Bool;
         END_STRUCT;
      END_STRUCT;
   END_VAR
   VAR
      ActualValues : Struct
         DateAndTime : DTL;
         DayOfYear : UInt;
      END_STRUCT;
      ShiftStatus { S7_SetPoint := 'True'} : "UDT_ShiftStatus";
      TimeTransformationRule { S7_SetPoint := 'True'} : TimeTransformationRule;
      Set_timezone_results { ExternalAccessible := 'False'; ExternalVisible := 'False'; ExternalWritable := 'False'} : Struct
         done { ExternalAccessible := 'False'; ExternalVisible := 'False'; ExternalWritable := 'False'} : Bool;
         busy { ExternalAccessible := 'False'; ExternalVisible := 'False'; ExternalWritable := 'False'} : Bool;
         error { ExternalAccessible := 'False'; ExternalVisible := 'False'; ExternalWritable := 'False'} : Bool;
         status { ExternalAccessible := 'False'; ExternalVisible := 'False'; ExternalWritable := 'False'} : Word;
      END_STRUCT;
   END_VAR
   VAR_TEMP
      i : Int;
      ui : UInt;
      actual_time : Time_Of_Day;
      dst : Bool;
   END_VAR
   VAR_TEMP   // added for the SCL form of the ladder/FBD networks
      _w1 : Bool;
      _w2 : Bool;
      _w3 : Bool;
      _w4 : Bool;
      _w5 : Bool;
      _w6 : Bool;
      _w7 : Bool;
      _w8 : Bool;
   END_VAR
BEGIN

REGION Network 1 (SCL)
   #TimeTransformationRule.Bias := -360;
   #TimeTransformationRule.DaylightBias := 0;
   #TimeTransformationRule.DaylightStartMonth := 3;
   #TimeTransformationRule.DaylightStartWeek := 5;
   #TimeTransformationRule.DaylightStartWeekday := 1;
   #TimeTransformationRule.DaylightStartHour := 2;
   #TimeTransformationRule.DaylightStartMinute := 0;
   #TimeTransformationRule.StandardStartMonth := 10;
   #TimeTransformationRule.StandardStartWeek := 5;
   #TimeTransformationRule.StandardStartWeekday := 1;
   #TimeTransformationRule.StandardStartHour := 3;
   #TimeTransformationRule.StandardStartMinute := 0;
END_REGION

REGION Network 2: Settings control
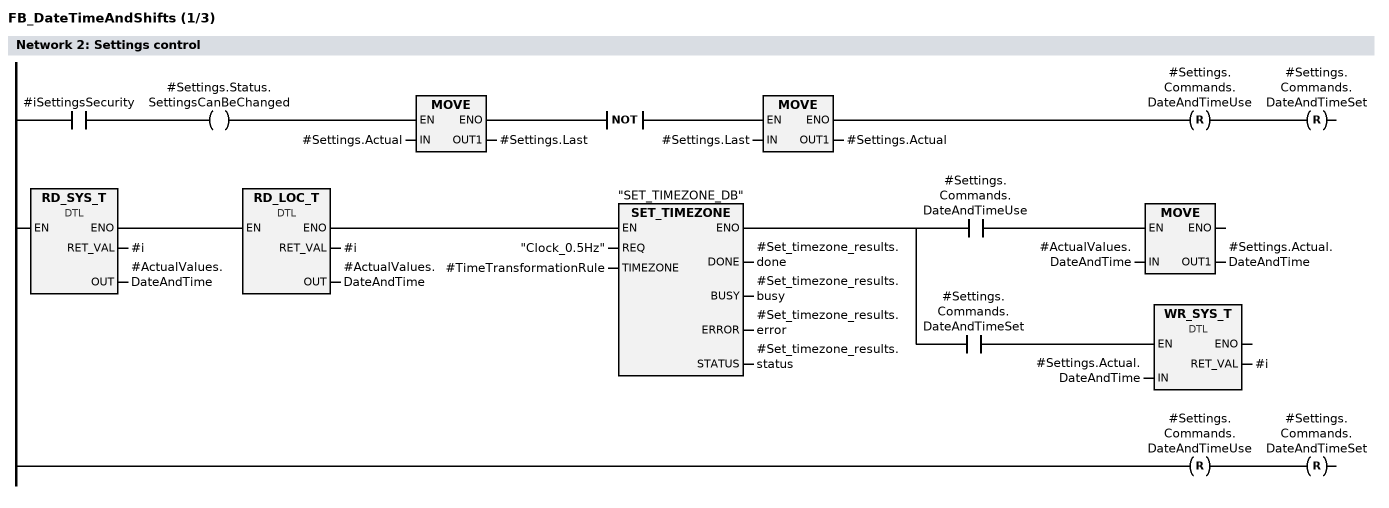
   RUNG wire#powerrail
      Contact( #iSettingsSecurity )
      Coil( #Settings.Status.SettingsCanBeChanged )
      Move(in := #Settings.Actual, out1 => #Settings.Last)
      Not()
      Move(in := #Settings.Last, out1 => #Settings.Actual)
      R_Coil( #Settings.Commands.DateAndTimeUse )
      R_Coil( #Settings.Commands.DateAndTimeSet )
   END_RUNG
   RUNG wire#powerrail
      { S7_Templates := "date_type := DTL" } RD_SYS_T(RET_VAL => #i, OUT => #ActualValues.DateAndTime)
      { S7_Templates := "date_type := DTL" } RD_LOC_T(RET_VAL => #i, OUT => #ActualValues.DateAndTime)
      "SET_TIMEZONE_DB".SET_TIMEZONE(REQ := "Clock_0.5Hz", TimeZone := #TimeTransformationRule, DONE => #Set_timezone_results.done, BUSY => #Set_timezone_results.busy, ERROR => #Set_timezone_results.error, STATUS => #Set_timezone_results.status)
      wire#w1
      Contact( #Settings.Commands.DateAndTimeUse )
      Move(in := #ActualValues.DateAndTime, out1 => #Settings.Actual.DateAndTime)
   END_RUNG
   RUNG wire#w1
      Contact( #Settings.Commands.DateAndTimeSet )
      { S7_Templates := "date_type := DTL" } WR_SYS_T(IN := #Settings.Actual.DateAndTime, RET_VAL => #i)
   END_RUNG
   RUNG wire#powerrail
      R_Coil( #Settings.Commands.DateAndTimeUse )
      R_Coil( #Settings.Commands.DateAndTimeSet )
   END_RUNG
   // the same network as SCL:
   #Settings.Status.SettingsCanBeChanged := #iSettingsSecurity;
   IF #iSettingsSecurity THEN #Settings.Last := #Settings.Actual; END_IF;
   IF NOT #iSettingsSecurity THEN
       #Settings.Actual := #Settings.Last;
       #Settings.Commands.DateAndTimeUse := FALSE;
       #Settings.Commands.DateAndTimeSet := FALSE;
   END_IF;
   #i := RD_SYS_T(OUT => #ActualValues.DateAndTime, ENO => #_w1);
   #i := RD_LOC_T(EN := #_w1, OUT => #ActualValues.DateAndTime, ENO => #_w2);
   "SET_TIMEZONE_DB"(EN := #_w2,   // SET_TIMEZONE
                     REQ := "Clock_0.5Hz",
                     TimeZone := #TimeTransformationRule,
                     DONE => #Set_timezone_results.done,
                     BUSY => #Set_timezone_results.busy,
                     ERROR => #Set_timezone_results.error,
                     STATUS => #Set_timezone_results.status,
                     ENO => #_w3);
   IF #_w3 AND #Settings.Commands.DateAndTimeUse THEN
       #Settings.Actual.DateAndTime := #ActualValues.DateAndTime;
   END_IF;
   IF #_w3 AND #Settings.Commands.DateAndTimeSet THEN
       #i := WR_SYS_T(IN := #Settings.Actual.DateAndTime);
   END_IF;
   #Settings.Commands.DateAndTimeUse := FALSE;
   #Settings.Commands.DateAndTimeSet := FALSE;
END_REGION

REGION Network 3: Day of year
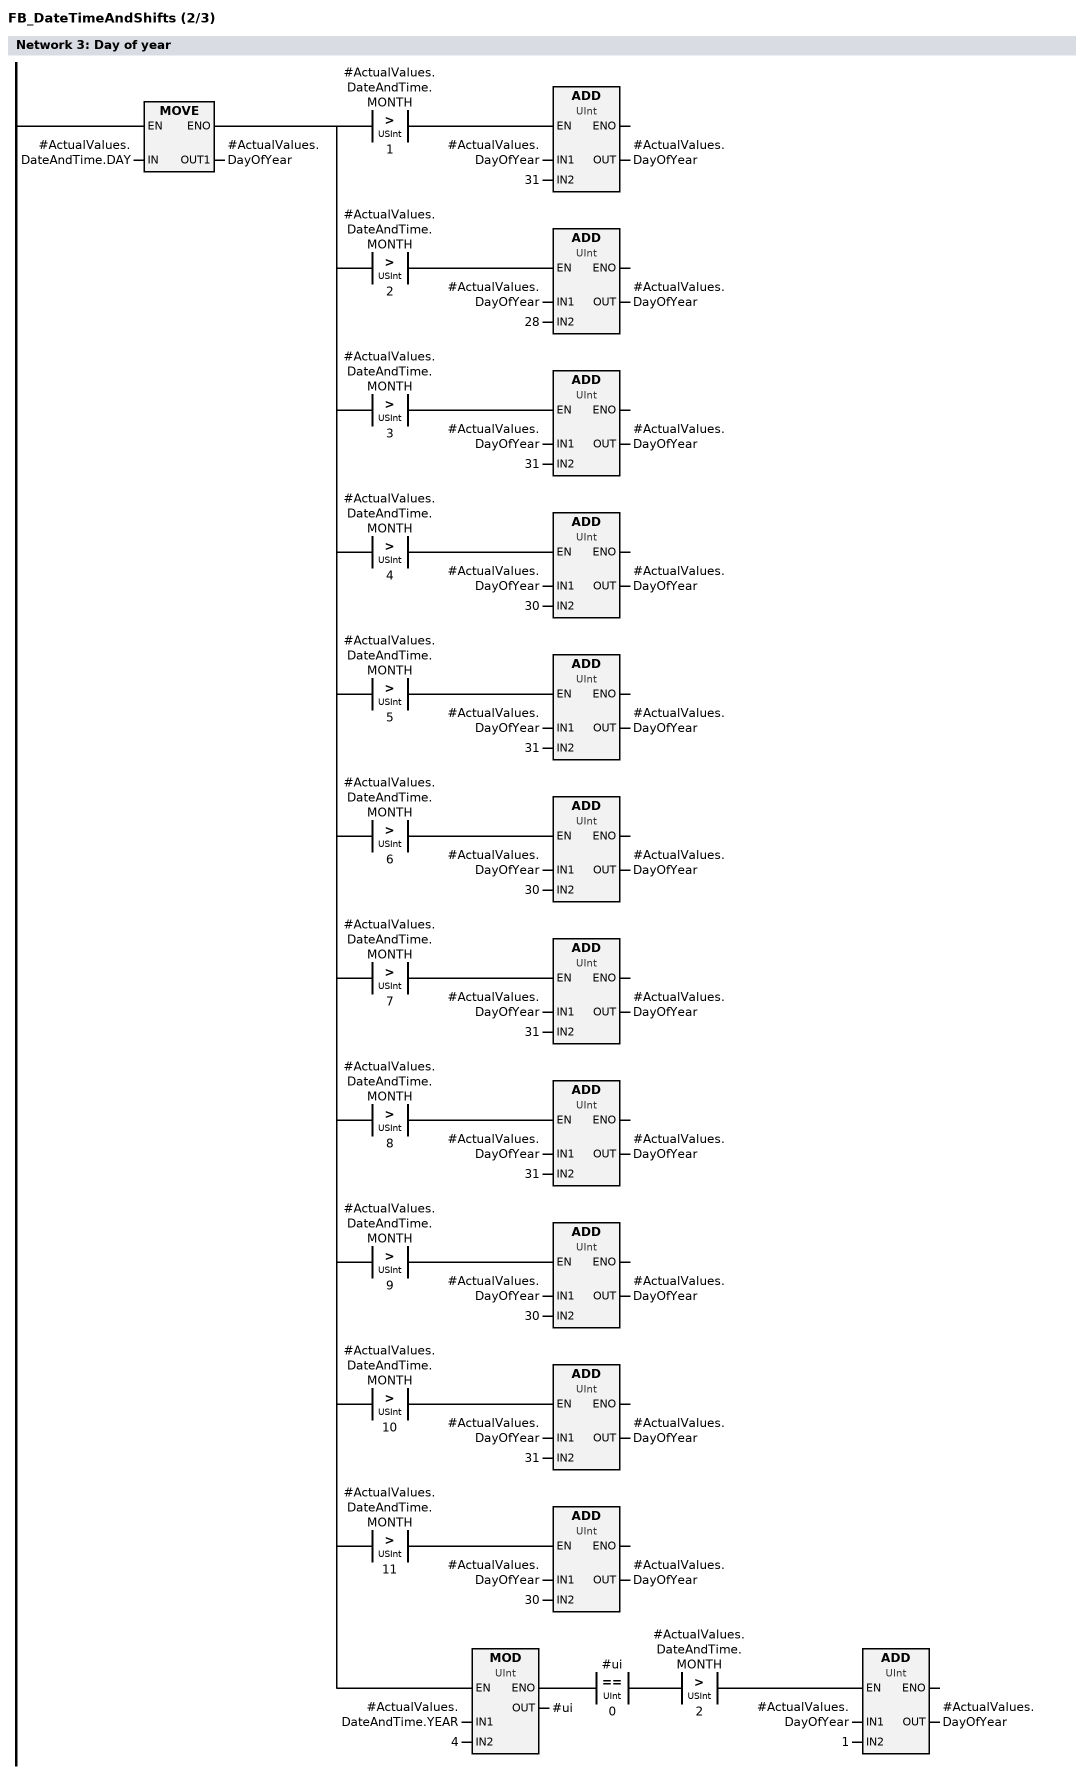
   RUNG wire#powerrail
      Move(in := #ActualValues.DateAndTime.DAY, out1 => #ActualValues.DayOfYear)
      wire#w1
      { S7_Templates := "SrcType := USInt" } GT_Contact(in1 := #ActualValues.DateAndTime.MONTH, in2 := 1)
      { S7_Templates := "SrcType := UInt" } Add(in1 := #ActualValues.DayOfYear, in2 := 31, out => #ActualValues.DayOfYear)
   END_RUNG
   RUNG wire#w1
      { S7_Templates := "SrcType := USInt" } GT_Contact(in1 := #ActualValues.DateAndTime.MONTH, in2 := 2)
      { S7_Templates := "SrcType := UInt" } Add(in1 := #ActualValues.DayOfYear, in2 := 28, out => #ActualValues.DayOfYear)
   END_RUNG
   RUNG wire#w1
      { S7_Templates := "SrcType := USInt" } GT_Contact(in1 := #ActualValues.DateAndTime.MONTH, in2 := 3)
      { S7_Templates := "SrcType := UInt" } Add(in1 := #ActualValues.DayOfYear, in2 := 31, out => #ActualValues.DayOfYear)
   END_RUNG
   RUNG wire#w1
      { S7_Templates := "SrcType := USInt" } GT_Contact(in1 := #ActualValues.DateAndTime.MONTH, in2 := 4)
      { S7_Templates := "SrcType := UInt" } Add(in1 := #ActualValues.DayOfYear, in2 := 30, out => #ActualValues.DayOfYear)
   END_RUNG
   RUNG wire#w1
      { S7_Templates := "SrcType := USInt" } GT_Contact(in1 := #ActualValues.DateAndTime.MONTH, in2 := 5)
      { S7_Templates := "SrcType := UInt" } Add(in1 := #ActualValues.DayOfYear, in2 := 31, out => #ActualValues.DayOfYear)
   END_RUNG
   RUNG wire#w1
      { S7_Templates := "SrcType := USInt" } GT_Contact(in1 := #ActualValues.DateAndTime.MONTH, in2 := 6)
      { S7_Templates := "SrcType := UInt" } Add(in1 := #ActualValues.DayOfYear, in2 := 30, out => #ActualValues.DayOfYear)
   END_RUNG
   RUNG wire#w1
      { S7_Templates := "SrcType := USInt" } GT_Contact(in1 := #ActualValues.DateAndTime.MONTH, in2 := 7)
      { S7_Templates := "SrcType := UInt" } Add(in1 := #ActualValues.DayOfYear, in2 := 31, out => #ActualValues.DayOfYear)
   END_RUNG
   RUNG wire#w1
      { S7_Templates := "SrcType := USInt" } GT_Contact(in1 := #ActualValues.DateAndTime.MONTH, in2 := 8)
      { S7_Templates := "SrcType := UInt" } Add(in1 := #ActualValues.DayOfYear, in2 := 31, out => #ActualValues.DayOfYear)
   END_RUNG
   RUNG wire#w1
      { S7_Templates := "SrcType := USInt" } GT_Contact(in1 := #ActualValues.DateAndTime.MONTH, in2 := 9)
      { S7_Templates := "SrcType := UInt" } Add(in1 := #ActualValues.DayOfYear, in2 := 30, out => #ActualValues.DayOfYear)
   END_RUNG
   RUNG wire#w1
      { S7_Templates := "SrcType := USInt" } GT_Contact(in1 := #ActualValues.DateAndTime.MONTH, in2 := 10)
      { S7_Templates := "SrcType := UInt" } Add(in1 := #ActualValues.DayOfYear, in2 := 31, out => #ActualValues.DayOfYear)
   END_RUNG
   RUNG wire#w1
      { S7_Templates := "SrcType := USInt" } GT_Contact(in1 := #ActualValues.DateAndTime.MONTH, in2 := 11)
      { S7_Templates := "SrcType := UInt" } Add(in1 := #ActualValues.DayOfYear, in2 := 30, out => #ActualValues.DayOfYear)
   END_RUNG
   RUNG wire#w1
      { S7_Templates := "SrcType := UInt" } Mod(in1 := #ActualValues.DateAndTime.YEAR, in2 := 4, out => #ui)
      { S7_Templates := "SrcType := UInt" } EQ_Contact(in1 := #ui, in2 := 0)
      { S7_Templates := "SrcType := USInt" } GT_Contact(in1 := #ActualValues.DateAndTime.MONTH, in2 := 2)
      { S7_Templates := "SrcType := UInt" } Add(in1 := #ActualValues.DayOfYear, in2 := 1, out => #ActualValues.DayOfYear)
   END_RUNG
   // the same network as SCL:
   #ActualValues.DayOfYear := #ActualValues.DateAndTime.DAY;
   IF #ActualValues.DateAndTime.MONTH > 1 THEN
       #ActualValues.DayOfYear := #ActualValues.DayOfYear + 31;
   END_IF;
   IF #ActualValues.DateAndTime.MONTH > 2 THEN
       #ActualValues.DayOfYear := #ActualValues.DayOfYear + 28;
   END_IF;
   IF #ActualValues.DateAndTime.MONTH > 3 THEN
       #ActualValues.DayOfYear := #ActualValues.DayOfYear + 31;
   END_IF;
   IF #ActualValues.DateAndTime.MONTH > 4 THEN
       #ActualValues.DayOfYear := #ActualValues.DayOfYear + 30;
   END_IF;
   IF #ActualValues.DateAndTime.MONTH > 5 THEN
       #ActualValues.DayOfYear := #ActualValues.DayOfYear + 31;
   END_IF;
   IF #ActualValues.DateAndTime.MONTH > 6 THEN
       #ActualValues.DayOfYear := #ActualValues.DayOfYear + 30;
   END_IF;
   IF #ActualValues.DateAndTime.MONTH > 7 THEN
       #ActualValues.DayOfYear := #ActualValues.DayOfYear + 31;
   END_IF;
   IF #ActualValues.DateAndTime.MONTH > 8 THEN
       #ActualValues.DayOfYear := #ActualValues.DayOfYear + 31;
   END_IF;
   IF #ActualValues.DateAndTime.MONTH > 9 THEN
       #ActualValues.DayOfYear := #ActualValues.DayOfYear + 30;
   END_IF;
   IF #ActualValues.DateAndTime.MONTH > 10 THEN
       #ActualValues.DayOfYear := #ActualValues.DayOfYear + 31;
   END_IF;
   IF #ActualValues.DateAndTime.MONTH > 11 THEN
       #ActualValues.DayOfYear := #ActualValues.DayOfYear + 30;
   END_IF;
   #ui := #ActualValues.DateAndTime.YEAR MOD 4;
   IF (#ui = 0) AND (#ActualValues.DateAndTime.MONTH > 2) THEN
       #ActualValues.DayOfYear := #ActualValues.DayOfYear + 1;
   END_IF;
END_REGION

REGION Network 4: Shifts
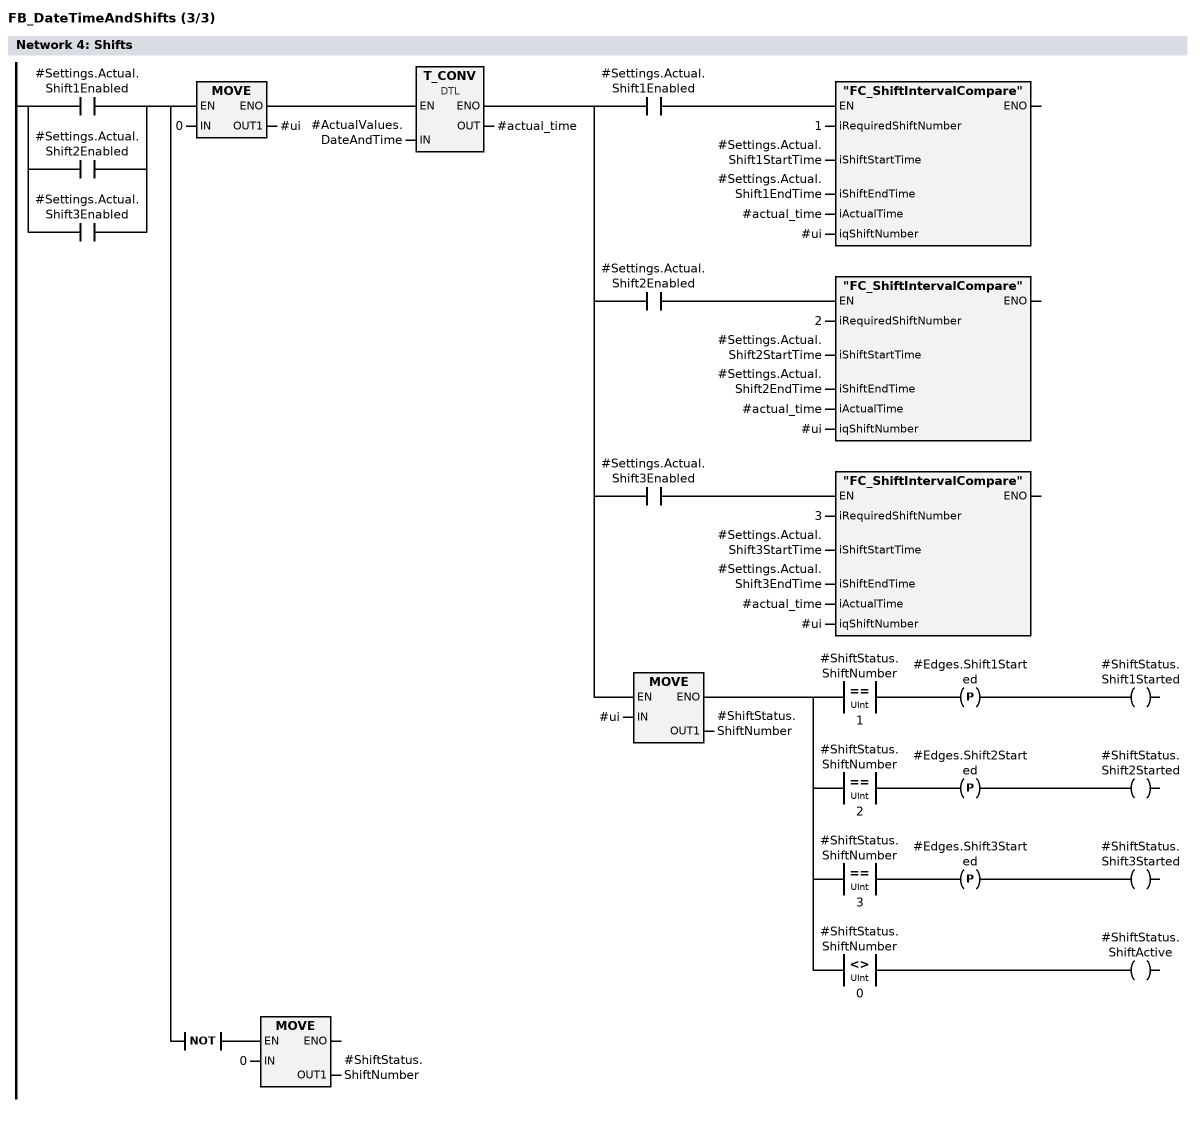
   RUNG wire#powerrail
      Contact( #Settings.Actual.Shift1Enabled )
      wire#w1
      Move(in := 0, out1 => #ui)
      { S7_Templates := "[src_type := DTL, dest_type := Time_Of_Day]" } T_CONV(IN := #ActualValues.DateAndTime, OUT => #actual_time)
      wire#w2
      Contact( #Settings.Actual.Shift1Enabled )
      "FC_ShiftIntervalCompare"(iRequiredShiftNumber := 1, iShiftStartTime := #Settings.Actual.Shift1StartTime, iShiftEndTime := #Settings.Actual.Shift1EndTime, iActualTime := #actual_time, iqShiftNumber := #ui)
   END_RUNG
   RUNG wire#powerrail
      Contact( #Settings.Actual.Shift2Enabled )
   END_RUNG wire#w1
   RUNG wire#powerrail
      Contact( #Settings.Actual.Shift3Enabled )
   END_RUNG wire#w1
   RUNG wire#w2
      Contact( #Settings.Actual.Shift2Enabled )
      "FC_ShiftIntervalCompare"(iRequiredShiftNumber := 2, iShiftStartTime := #Settings.Actual.Shift2StartTime, iShiftEndTime := #Settings.Actual.Shift2EndTime, iActualTime := #actual_time, iqShiftNumber := #ui)
   END_RUNG
   RUNG wire#w2
      Contact( #Settings.Actual.Shift3Enabled )
      "FC_ShiftIntervalCompare"(iRequiredShiftNumber := 3, iShiftStartTime := #Settings.Actual.Shift3StartTime, iShiftEndTime := #Settings.Actual.Shift3EndTime, iActualTime := #actual_time, iqShiftNumber := #ui)
   END_RUNG
   RUNG wire#w2
      Move(in := #ui, out1 => #ShiftStatus.ShiftNumber)
      wire#w3
      { S7_Templates := "SrcType := UInt" } EQ_Contact(in1 := #ShiftStatus.ShiftNumber, in2 := 1)
      P_Trig( #Edges.Shift1Started )
      Coil( #ShiftStatus.Shift1Started )
   END_RUNG
   RUNG wire#w3
      { S7_Templates := "SrcType := UInt" } EQ_Contact(in1 := #ShiftStatus.ShiftNumber, in2 := 2)
      P_Trig( #Edges.Shift2Started )
      Coil( #ShiftStatus.Shift2Started )
   END_RUNG
   RUNG wire#w3
      { S7_Templates := "SrcType := UInt" } EQ_Contact(in1 := #ShiftStatus.ShiftNumber, in2 := 3)
      P_Trig( #Edges.Shift3Started )
      Coil( #ShiftStatus.Shift3Started )
   END_RUNG
   RUNG wire#w3
      { S7_Templates := "SrcType := UInt" } NE_Contact(in1 := #ShiftStatus.ShiftNumber, in2 := 0)
      Coil( #ShiftStatus.ShiftActive )
   END_RUNG
   RUNG wire#w1
      Not()
      Move(in := 0, out1 => #ShiftStatus.ShiftNumber)
   END_RUNG
   // the same network as SCL:
   #_w1 := #Settings.Actual.Shift1Enabled OR #Settings.Actual.Shift2Enabled OR #Settings.Actual.Shift3Enabled;
   IF #_w1 THEN #ui := 0; END_IF;
   T_CONV(EN := #_w1, IN := #ActualValues.DateAndTime, OUT => #actual_time, ENO => #_w2);
   IF #_w2 AND #Settings.Actual.Shift1Enabled THEN
       "FC_ShiftIntervalCompare"(iRequiredShiftNumber := 1,
                               iShiftStartTime := #Settings.Actual.Shift1StartTime,
                               iShiftEndTime := #Settings.Actual.Shift1EndTime,
                               iActualTime := #actual_time,
                               iqShiftNumber := #ui);
   END_IF;
   IF #_w2 AND #Settings.Actual.Shift2Enabled THEN
       "FC_ShiftIntervalCompare"(iRequiredShiftNumber := 2,
                               iShiftStartTime := #Settings.Actual.Shift2StartTime,
                               iShiftEndTime := #Settings.Actual.Shift2EndTime,
                               iActualTime := #actual_time,
                               iqShiftNumber := #ui);
   END_IF;
   IF #_w2 AND #Settings.Actual.Shift3Enabled THEN
       "FC_ShiftIntervalCompare"(iRequiredShiftNumber := 3,
                               iShiftStartTime := #Settings.Actual.Shift3StartTime,
                               iShiftEndTime := #Settings.Actual.Shift3EndTime,
                               iActualTime := #actual_time,
                               iqShiftNumber := #ui);
   END_IF;
   IF #_w2 THEN #ShiftStatus.ShiftNumber := #ui; END_IF;
   #_w3 := #_w2 AND (#ShiftStatus.ShiftNumber = 1);
   #_w4 := #_w3 AND NOT #Edges.Shift1Started;   // rising edge
   #Edges.Shift1Started := #_w3;
   #ShiftStatus.Shift1Started := #_w4;
   #_w5 := #_w2 AND (#ShiftStatus.ShiftNumber = 2);
   #_w6 := #_w5 AND NOT #Edges.Shift2Started;   // rising edge
   #Edges.Shift2Started := #_w5;
   #ShiftStatus.Shift2Started := #_w6;
   #_w7 := #_w2 AND (#ShiftStatus.ShiftNumber = 3);
   #_w8 := #_w7 AND NOT #Edges.Shift3Started;   // rising edge
   #Edges.Shift3Started := #_w7;
   #ShiftStatus.Shift3Started := #_w8;
   #ShiftStatus.ShiftActive := #_w2 AND (#ShiftStatus.ShiftNumber <> 0);
   IF NOT #_w1 THEN #ShiftStatus.ShiftNumber := 0; END_IF;
END_REGION
END_FUNCTION_BLOCK

FUNCTION "FC_ShiftIntervalCompare" : Void   // FC5010, LAD
{ S7_Optimized_Access := 'TRUE' }
VERSION : 0.1
// stored: AutoNumber false, IsIECCheckEnabled false, SetENOAutomatically false, UDAEnableTagReadback false
   VAR_INPUT
      iRequiredShiftNumber : UInt;
      iShiftStartTime : Time_Of_Day;
      iShiftEndTime : Time_Of_Day;
      iActualTime : Time_Of_Day;
   END_VAR
   VAR_IN_OUT
      iqShiftNumber : UInt;
   END_VAR
   VAR_TEMP
      midnight_time : Time_Of_Day;
      morning_time : Time_Of_Day;
      interval_in_two_days : Bool;
   END_VAR
BEGIN

REGION Network 1: Shift interval compare
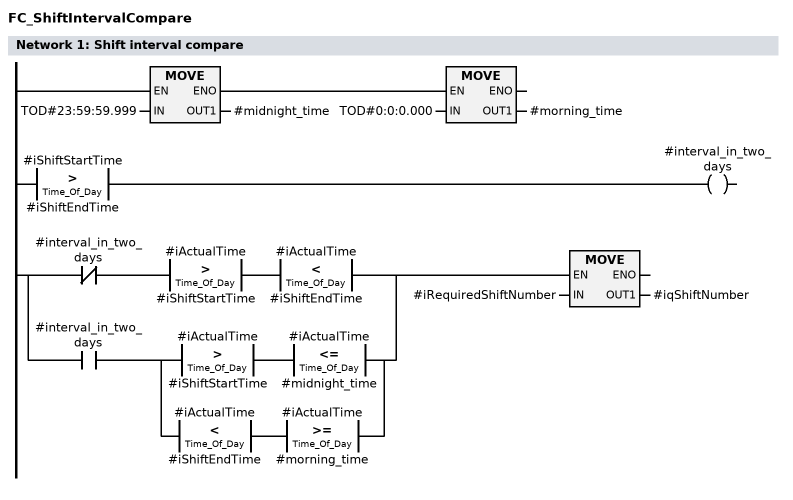
   RUNG wire#powerrail
      Move(in := TOD#23:59:59.999, out1 => #midnight_time)
      Move(in := TOD#0:0:0.000, out1 => #morning_time)
   END_RUNG
   RUNG wire#powerrail
      { S7_Templates := "SrcType := Time_Of_Day" } GT_Contact(in1 := #iShiftStartTime, in2 := #iShiftEndTime)
      Coil( #interval_in_two_days )
   END_RUNG
   RUNG wire#powerrail
      I_Contact( #interval_in_two_days )
      { S7_Templates := "SrcType := Time_Of_Day" } GT_Contact(in1 := #iActualTime, in2 := #iShiftStartTime)
      { S7_Templates := "SrcType := Time_Of_Day" } LT_Contact(in1 := #iActualTime, in2 := #iShiftEndTime)
      wire#w1
      Move(in := #iRequiredShiftNumber, out1 => #iqShiftNumber)
   END_RUNG
   RUNG wire#powerrail
      Contact( #interval_in_two_days )
      wire#w2
      { S7_Templates := "SrcType := Time_Of_Day" } GT_Contact(in1 := #iActualTime, in2 := #iShiftStartTime)
      { S7_Templates := "SrcType := Time_Of_Day" } LE_Contact(in1 := #iActualTime, in2 := #midnight_time)
   END_RUNG wire#w1
   RUNG wire#w2
      { S7_Templates := "SrcType := Time_Of_Day" } LT_Contact(in1 := #iActualTime, in2 := #iShiftEndTime)
      { S7_Templates := "SrcType := Time_Of_Day" } GE_Contact(in1 := #iActualTime, in2 := #morning_time)
   END_RUNG wire#w1
   // the same network as SCL:
   #midnight_time := TOD#23:59:59.999;
   #morning_time := TOD#0:0:0.000;
   #interval_in_two_days := #iShiftStartTime > #iShiftEndTime;
   IF (NOT #interval_in_two_days AND (#iActualTime > #iShiftStartTime) AND (#iActualTime < #iShiftEndTime)) OR (#interval_in_two_days AND (((#iActualTime > #iShiftStartTime) AND (#iActualTime <= #midnight_time)) OR ((#iActualTime < #iShiftEndTime) AND (#iActualTime >= #morning_time)))) THEN
       #iqShiftNumber := #iRequiredShiftNumber;
   END_IF;
END_REGION
END_FUNCTION

FUNCTION "FC_ProductionProgram" : Void   // FC6100, LAD
{ S7_Optimized_Access := 'TRUE' }
VERSION : 0.1
// stored: AutoNumber false, IsIECCheckEnabled false, SetENOAutomatically false, UDAEnableTagReadback false
   VAR_INPUT
      iSettingsSecurity : Bool;
      iBlinker : Bool;
   END_VAR
BEGIN

REGION Network 1 (SCL): Production program edit
   //Actual program
   IF "DB_ProductionProgramActual".ProgrammNumber < 1 OR "DB_ProductionProgramActual".ProgrammNumber > "NumberOfProductionPrograms" THEN
       "DB_ProductionProgramActual".ProgrammNumber := 1;
   END_IF;
   "DB_ProductionProgramActual".Program := "DB_ProductionProgramList".Program["DB_ProductionProgramActual".ProgrammNumber];
   "DB_ProductionProgramActual".Program.CupformingParametersRight.ApproachForce := "DB_ProductionProgramActual".Program.CupformingParametersLeft.ApproachForce;
   "DB_ProductionProgramActual".Program.CupformingParametersRight.FinalForce := "DB_ProductionProgramActual".Program.CupformingParametersLeft.FinalForce;

   //Program to edit: Number limits
   IF "DB_ProductionProgramEdit".Commands.ProgramEdit.Number < 1 THEN
       "DB_ProductionProgramEdit".Commands.ProgramEdit.Number := 1;
   END_IF;

   IF "DB_ProductionProgramEdit".Commands.ProgramEdit.Number > "NumberOfProductionPrograms" THEN
       "DB_ProductionProgramEdit".Commands.ProgramEdit.Number := "NumberOfProductionPrograms";
   END_IF;

   //Program to edit: Number changed
   "DB_ProductionProgramEdit".Commands.ProgramEdit.NumberChanged := FALSE;
   IF "DB_ProductionProgramEdit".Commands.ProgramEdit.Number <> "DB_ProductionProgramEdit".Commands.ProgramEdit.NumberLast THEN
       "DB_ProductionProgramEdit".Commands.ProgramEdit.NumberLast := "DB_ProductionProgramEdit".Commands.ProgramEdit.Number;
       "DB_ProductionProgramEdit".Commands.ProgramEdit.NumberChanged := TRUE;
   END_IF;

   //Program to edit: Load
   IF #iSettingsSecurity = FALSE OR
       "DB_ProductionProgramEdit".Commands.ProgramEdit.NumberChanged = TRUE OR
       "DB_ProductionProgramEdit".Commands.ProgramEdit.LoadAll = TRUE THEN
       "DB_ProductionProgramEdit".Commands.ProgramEdit.Commands := 1;
   END_IF;

   IF "DB_ProductionProgramEdit".Commands.ProgramEdit.Commands = 1 THEN
       "DB_ProductionProgramEdit".ProgramEdit := "DB_ProductionProgramList".Program["DB_ProductionProgramEdit".Commands.ProgramEdit.Number];
   END_IF;

   //Product to edit: Number limits
   IF "DB_ProductionProgramEdit".Commands.ProgramEdit.NumberChanged = TRUE OR
       "DB_ProductionProgramEdit".Commands.ProgramEdit.LoadAll = TRUE THEN
       "DB_ProductionProgramEdit".Commands.ProductEdit.Number := 1;
   END_IF;

   IF "DB_ProductionProgramEdit".Commands.ProductEdit.Number < 1 THEN
       "DB_ProductionProgramEdit".Commands.ProductEdit.Number := 1;
   END_IF;

   IF "DB_ProductionProgramEdit".Commands.ProductEdit.Number > "NumberOfProductionProducts" THEN
       "DB_ProductionProgramEdit".Commands.ProductEdit.Number := "NumberOfProductionProducts";
   END_IF;

   //Product to edit: Number changed
   "DB_ProductionProgramEdit".Commands.ProductEdit.NumberChanged := FALSE;
   IF "DB_ProductionProgramEdit".Commands.ProductEdit.Number <> "DB_ProductionProgramEdit".Commands.ProductEdit.NumberLast THEN
       "DB_ProductionProgramEdit".Commands.ProductEdit.NumberLast := "DB_ProductionProgramEdit".Commands.ProductEdit.Number;
       "DB_ProductionProgramEdit".Commands.ProductEdit.NumberChanged := TRUE;
   END_IF;


   //Position to edit: Number limits
   IF "DB_ProductionProgramEdit".Commands.ProgramEdit.NumberChanged = TRUE OR
       "DB_ProductionProgramEdit".Commands.ProgramEdit.LoadAll = TRUE OR
       "DB_ProductionProgramEdit".Commands.ProductEdit.NumberChanged = TRUE THEN
       "DB_ProductionProgramEdit".Commands.PositionEdit.Number := 1;
   END_IF;

   IF "DB_ProductionProgramEdit".Commands.PositionEdit.Number < 1 THEN
       "DB_ProductionProgramEdit".Commands.PositionEdit.Number := 1;
   END_IF;

   //Position to edit: Number changed
   "DB_ProductionProgramEdit".Commands.PositionEdit.NumberChanged := FALSE;
   IF "DB_ProductionProgramEdit".Commands.PositionEdit.Number <> "DB_ProductionProgramEdit".Commands.PositionEdit.NumberLast THEN
       "DB_ProductionProgramEdit".Commands.PositionEdit.NumberLast := "DB_ProductionProgramEdit".Commands.PositionEdit.Number;
       "DB_ProductionProgramEdit".Commands.PositionEdit.NumberChanged := TRUE;
   END_IF;

   //Position to edit: Load
   "DB_ProductionProgramEdit".Commands.PositionEdit.Load := FALSE;
   IF "DB_ProductionProgramEdit".Commands.ProgramEdit.Commands = 1 OR
       "DB_ProductionProgramEdit".Commands.ProductEdit.NumberChanged = TRUE OR
       "DB_ProductionProgramEdit".Commands.PositionEdit.NumberChanged = TRUE THEN
       "DB_ProductionProgramEdit".Commands.PositionEdit.Load := TRUE;
   END_IF;

   //Save program
   IF "DB_ProductionProgramEdit".Commands.ProgramEdit.Commands = 2 THEN
       "DB_ProductionProgramList".Program["DB_ProductionProgramEdit".Commands.ProgramEdit.Number] := "DB_ProductionProgramEdit".ProgramEdit;
       "READER_MODEL".PRODUCT["DB_ProductionProgramEdit".Commands.ProgramEdit.Number] := "READER_MODEL_ACTUAL".EDIT;
   END_IF;

   //Copy program
   IF "DB_ProductionProgramEdit".Commands.ProgramEdit.Commands = 3 THEN
       "DB_ProductionProgramEdit".ProgramInBox := "DB_ProductionProgramEdit".ProgramEdit;
       "DB_ProductionProgramEdit".Commands.ProgramEdit.NumberInBox := "DB_ProductionProgramEdit".Commands.ProgramEdit.Number;
       "READER_MODEL_ACTUAL".IN_BOX := "READER_MODEL_ACTUAL".EDIT;
   END_IF;

   //Paste program
   IF "DB_ProductionProgramEdit".Commands.ProgramEdit.Commands = 4 THEN
       "DB_ProductionProgramEdit".ProgramEdit := "DB_ProductionProgramEdit".ProgramInBox;
       "READER_MODEL_ACTUAL".EDIT := "READER_MODEL_ACTUAL".IN_BOX;
   END_IF;

   //Delete program
   IF "DB_ProductionProgramEdit".Commands.ProgramEdit.Commands = 5 THEN
       "DB_ProductionProgramEdit".ProgramEdit := "DB_ProductionProgramEdit".ProgramEmpty;
   END_IF;

   //Program to edit: Check if it was changed
   "DB_ProductionProgramEdit".Commands.ProgramEdit.ProgramChanged := FALSE;
   IF "DB_ProductionProgramEdit".ProgramEdit <> "DB_ProductionProgramList".Program["DB_ProductionProgramEdit".Commands.ProgramEdit.Number]
       OR  "READER_MODEL_ACTUAL".EDIT <> "READER_MODEL".PRODUCT["DB_ProductionProgramEdit".Commands.ProgramEdit.Number]THEN
       "DB_ProductionProgramEdit".Commands.ProgramEdit.ProgramChanged := TRUE;
   END_IF;
END_REGION

REGION Network 2: Command status
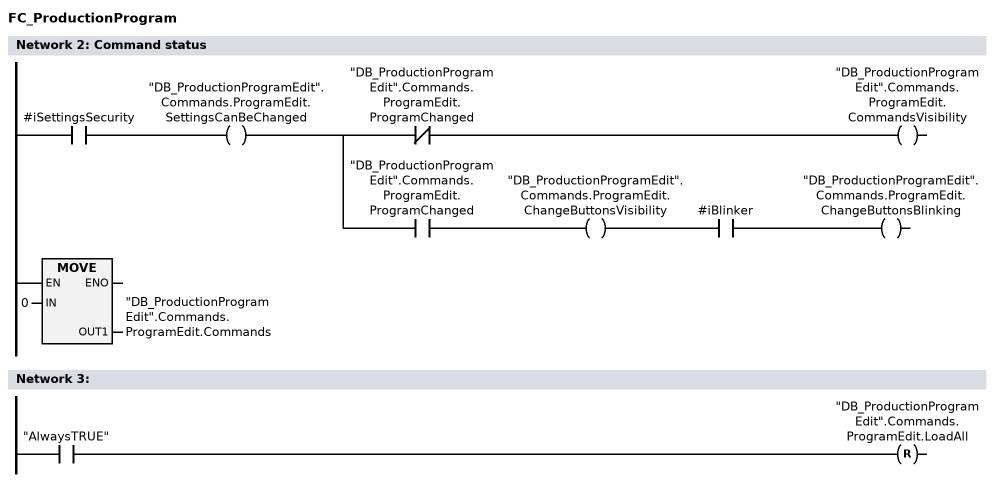
   RUNG wire#powerrail
      Contact( #iSettingsSecurity )
      Coil( "DB_ProductionProgramEdit".Commands.ProgramEdit.SettingsCanBeChanged )
      wire#w1
      I_Contact( "DB_ProductionProgramEdit".Commands.ProgramEdit.ProgramChanged )
      Coil( "DB_ProductionProgramEdit".Commands.ProgramEdit.CommandsVisibility )
   END_RUNG
   RUNG wire#w1
      Contact( "DB_ProductionProgramEdit".Commands.ProgramEdit.ProgramChanged )
      Coil( "DB_ProductionProgramEdit".Commands.ProgramEdit.ChangeButtonsVisibility )
      Contact( #iBlinker )
      Coil( "DB_ProductionProgramEdit".Commands.ProgramEdit.ChangeButtonsBlinking )
   END_RUNG
   RUNG wire#powerrail
      Move(in := 0, out1 => "DB_ProductionProgramEdit".Commands.ProgramEdit.Commands)
   END_RUNG
   // the same network as SCL:
   "DB_ProductionProgramEdit".Commands.ProgramEdit.SettingsCanBeChanged := #iSettingsSecurity;
   "DB_ProductionProgramEdit".Commands.ProgramEdit.CommandsVisibility := #iSettingsSecurity AND NOT "DB_ProductionProgramEdit".Commands.ProgramEdit.ProgramChanged;
   "DB_ProductionProgramEdit".Commands.ProgramEdit.ChangeButtonsVisibility := #iSettingsSecurity AND "DB_ProductionProgramEdit".Commands.ProgramEdit.ProgramChanged;
   "DB_ProductionProgramEdit".Commands.ProgramEdit.ChangeButtonsBlinking := "DB_ProductionProgramEdit".Commands.ProgramEdit.ChangeButtonsVisibility AND #iBlinker;
   "DB_ProductionProgramEdit".Commands.ProgramEdit.Commands := 0;
END_REGION

REGION Network 3
   RUNG wire#powerrail
      Contact( "AlwaysTRUE" )
      R_Coil( "DB_ProductionProgramEdit".Commands.ProgramEdit.LoadAll )
   END_RUNG
   // the same network as SCL:
   IF "AlwaysTRUE" THEN "DB_ProductionProgramEdit".Commands.ProgramEdit.LoadAll := FALSE; END_IF;
END_REGION
END_FUNCTION

FUNCTION_BLOCK "FB_Devices"   // FB5100, LAD
{ S7_Optimized_Access := 'TRUE' }
VERSION : 0.1
// stored: AutoNumber false, IsIECCheckEnabled false, IsRetainMemResEnabled false, MemoryReserve 100, SetENOAutomatically false, UDAEnableTagReadback false
   VAR
      ServiceDoors_Instance_1 { S7_SetPoint := 'True'} : "serviceDoor";
      ServiceDoors_Instance_2 { S7_SetPoint := 'True'} : "serviceDoor";
      R_TRIG_Instance { S7_SetPoint := 'True'} : R_TRIG;
      HydraulicActive { S7_SetPoint := 'True'} : Bool;
      HydraulicActiveOffMem : Bool;
      HydraulicOnMem : Bool;
      IEC_Timer_0_Instance { S7_SetPoint := 'True'} : TON_TIME;
      IEC_Timer_0_Instance_1 { S7_SetPoint := 'True'} : TON_TIME;
      FB_TurnTable_Instance { S7_SetPoint := 'True'} : "FB_TurnTable";
      F_TRIG_Instance { S7_SetPoint := 'True'} : F_TRIG;
      edges { S7_SetPoint := 'True'} : Array[1..6] of Bool;
      ManualCommandOld : Int;
      R_TRIG_Instance_1 { S7_SetPoint := 'True'} : R_TRIG;
      R_TRIG_Instance_2 { S7_SetPoint := 'True'} : R_TRIG;
      R_TRIG_Instance_3 { S7_SetPoint := 'True'} : R_TRIG;
      R_TRIG_Instance_4 { S7_SetPoint := 'True'} : R_TRIG;
      R_TRIG_Instance_6 { S7_SetPoint := 'True'} : R_TRIG;
      R_TRIG_Instance_7 { S7_SetPoint := 'True'} : R_TRIG;
      R_TRIG_Instance_8 { S7_SetPoint := 'True'} : R_TRIG;
      R_TRIG_Instance_5 { S7_SetPoint := 'True'} : R_TRIG;
      edgesFitting : Array[1..4] of Bool;
      R_TRIG_V240Wp { S7_SetPoint := 'True'} : R_TRIG;
      R_TRIG_V240Bp { S7_SetPoint := 'True'} : R_TRIG;
      ReaderKeyence_Instance { S7_SetPoint := 'True'} : "ReaderKeyence";
      IEC_Timer_0_Instance_2 { S7_SetPoint := 'True'} : TON_TIME;
      FriedrichUnit1_Instance { S7_SetPoint := 'True'} : "FriedrichUnit";
      FriedrichUnit2_Instance { S7_SetPoint := 'True'} : "FriedrichUnit";
      Trig1 { S7_SetPoint := 'True'} : R_TRIG;
      Trig2 { S7_SetPoint := 'True'} : R_TRIG;
      Trig3 { S7_SetPoint := 'True'} : R_TRIG;
      Trig4 { S7_SetPoint := 'True'} : R_TRIG;
      Camera_CAM1 { S7_SetPoint := 'True'} : "Camera";
      Camera_CAM2 { S7_SetPoint := 'True'} : "Camera";
      Camera_CAM3 { S7_SetPoint := 'True'} : "Camera";
      Camera_CAM4 { S7_SetPoint := 'True'} : "Camera";
      RivetingCycleLeft_Instance { S7_SetPoint := 'True'} : "RivetingCycle";
      RivetingCycleRight_Instance { S7_SetPoint := 'True'} : "RivetingCycle";
   END_VAR
   VAR_TEMP
      posTemp : "UDT_PositionData";
      i : Int;
   END_VAR
   VAR_TEMP   // added for the SCL form of the ladder/FBD networks
      _w1 : Bool;
      _w2 : Bool;
      _w3 : Bool;
   END_VAR
BEGIN

REGION Network 1: Diagnostic fieldbus devices
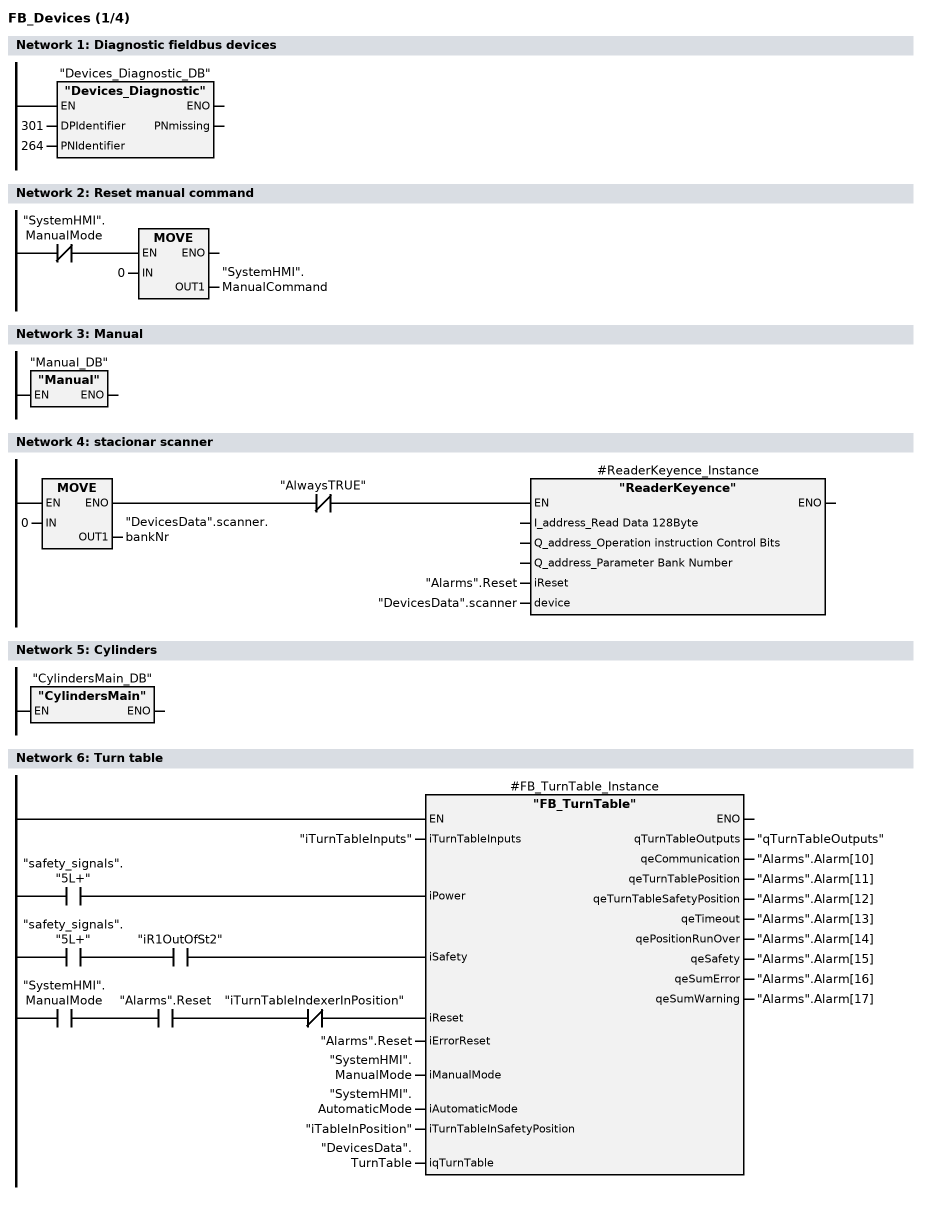
   RUNG wire#powerrail
      "Devices_Diagnostic_DB"(DPIdentifier := 301, PNIdentifier := 264, PNmissing =>)
   END_RUNG
   // the same network as SCL:
   "Devices_Diagnostic_DB"(DPIdentifier := 301, PNIdentifier := 264);   // "Devices_Diagnostic"
END_REGION

REGION Network 2: Reset manual command
   RUNG wire#powerrail
      I_Contact( "SystemHMI".ManualMode )
      Move(in := 0, out1 => "SystemHMI".ManualCommand)
   END_RUNG
   // the same network as SCL:
   IF NOT "SystemHMI".ManualMode THEN "SystemHMI".ManualCommand := 0; END_IF;
END_REGION

REGION Network 3: Manual
   RUNG wire#powerrail
      "Manual_DB"()
   END_RUNG
   // the same network as SCL:
   "Manual_DB"();   // "Manual"
END_REGION

REGION Network 4: stacionar scanner
   RUNG wire#powerrail
      Move(in := 0, out1 => "DevicesData".scanner.bankNr)
      I_Contact( "AlwaysTRUE" )
      #ReaderKeyence_Instance("I_address_Read Data 128Byte" :=, "Q_address_Operation instruction Control Bits" :=, "Q_address_Parameter Bank Number" :=, iReset := "Alarms".Reset, device := "DevicesData".scanner)
   END_RUNG
   // the same network as SCL:
   "DevicesData".scanner.bankNr := 0;
   IF NOT "AlwaysTRUE" THEN
       #ReaderKeyence_Instance(iReset := "Alarms".Reset, device := "DevicesData".scanner);   // "ReaderKeyence"
   END_IF;
END_REGION

REGION Network 5: Cylinders
   RUNG wire#powerrail
      "CylindersMain_DB"()
   END_RUNG
   // the same network as SCL:
   "CylindersMain_DB"();   // "CylindersMain"
END_REGION

REGION Network 6: Turn table
   RUNG wire#powerrail
      #FB_TurnTable_Instance(iPower := wire#w1, iSafety := wire#w2, iReset := wire#w3, iTurnTableInputs := "iTurnTableInputs", iErrorReset := "Alarms".Reset, iManualMode := "SystemHMI".ManualMode, iAutomaticMode := "SystemHMI".AutomaticMode, iTurnTableInSafetyPosition := "iTableInPosition", iqTurnTable := "DevicesData".TurnTable, qTurnTableOutputs => "qTurnTableOutputs", qeCommunication => "Alarms".Alarm[10], qeTurnTablePosition => "Alarms".Alarm[11], qeTurnTableSafetyPosition => "Alarms".Alarm[12], qeTimeout => "Alarms".Alarm[13], qePositionRunOver => "Alarms".Alarm[14], qeSafety => "Alarms".Alarm[15], qeSumError => "Alarms".Alarm[16], qeSumWarning => "Alarms".Alarm[17])
   END_RUNG
   RUNG wire#powerrail
      Contact( "safety_signals"."5L+" )
   END_RUNG wire#w1
   RUNG wire#powerrail
      Contact( "safety_signals"."5L+" )
      Contact( "iR1OutOfSt2" )
   END_RUNG wire#w2
   RUNG wire#powerrail
      Contact( "SystemHMI".ManualMode )
      Contact( "Alarms".Reset )
      I_Contact( "iTurnTableIndexerInPosition" )
   END_RUNG wire#w3
   // the same network as SCL:
   #FB_TurnTable_Instance(iTurnTableInputs := "iTurnTableInputs",   // "FB_TurnTable"
                          iPower := "safety_signals"."5L+",
                          iSafety := "safety_signals"."5L+" AND "iR1OutOfSt2",
                          iReset := "SystemHMI".ManualMode AND "Alarms".Reset AND NOT "iTurnTableIndexerInPosition",
                          iErrorReset := "Alarms".Reset,
                          iManualMode := "SystemHMI".ManualMode,
                          iAutomaticMode := "SystemHMI".AutomaticMode,
                          iTurnTableInSafetyPosition := "iTableInPosition",
                          iqTurnTable := "DevicesData".TurnTable,
                          qTurnTableOutputs => "qTurnTableOutputs",
                          qeCommunication => "Alarms".Alarm[10],
                          qeTurnTablePosition => "Alarms".Alarm[11],
                          qeTurnTableSafetyPosition => "Alarms".Alarm[12],
                          qeTimeout => "Alarms".Alarm[13],
                          qePositionRunOver => "Alarms".Alarm[14],
                          qeSafety => "Alarms".Alarm[15],
                          qeSumError => "Alarms".Alarm[16],
                          qeSumWarning => "Alarms".Alarm[17]);
END_REGION

REGION Network 7: Handle table positions
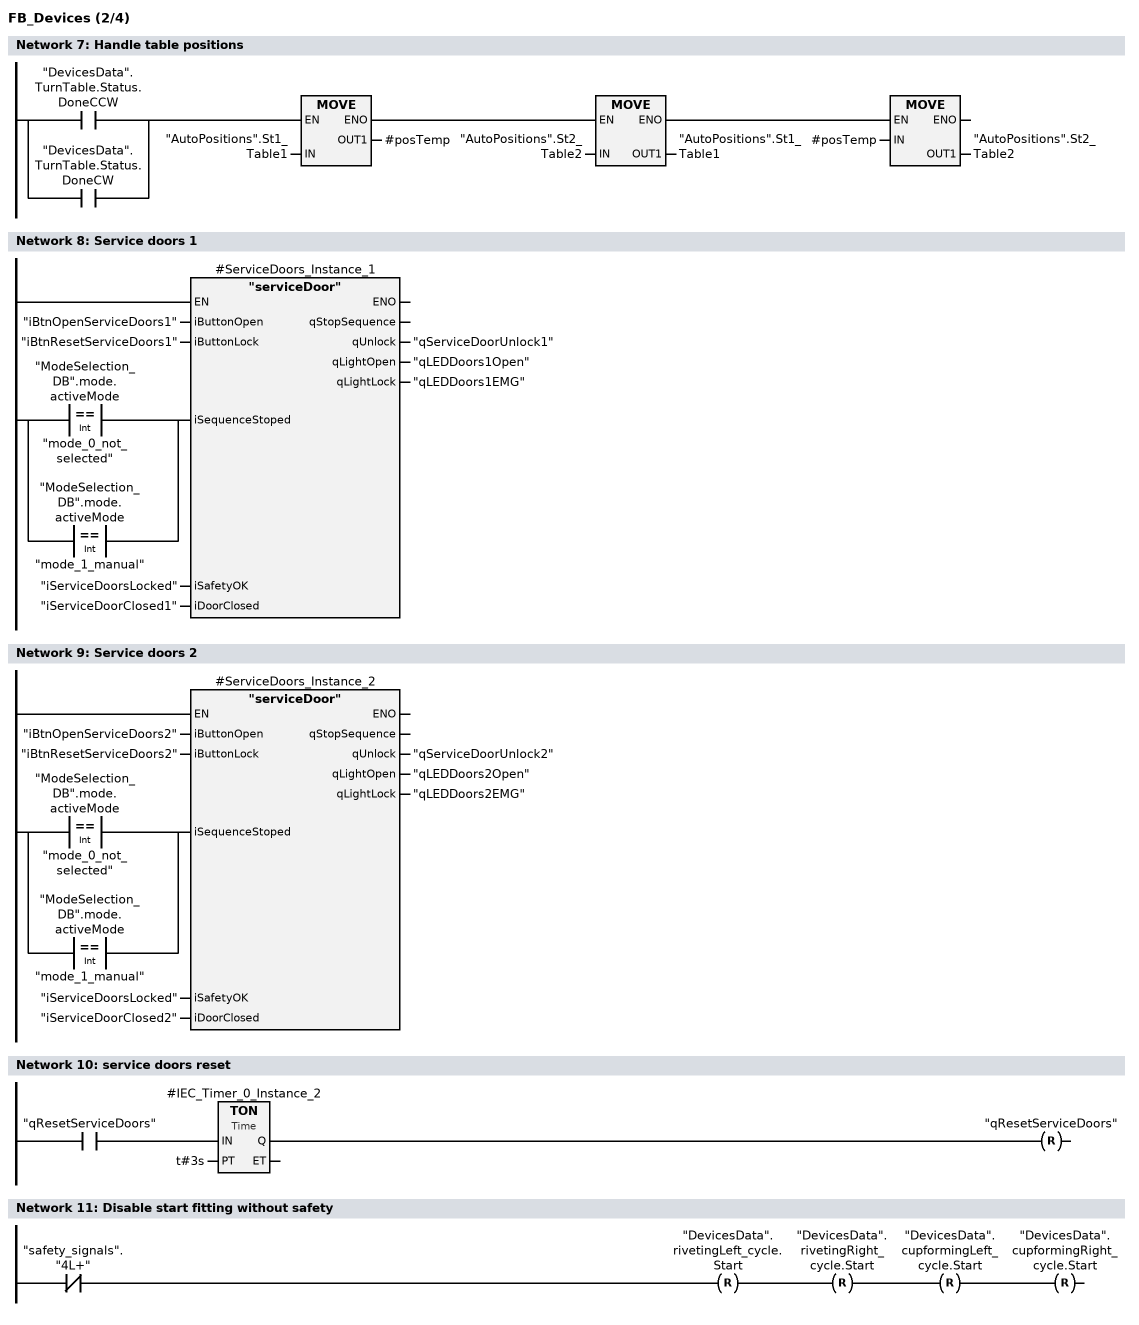
   RUNG wire#powerrail
      Contact( "DevicesData".TurnTable.Status.DoneCCW )
      wire#w1
      Move(in := "AutoPositions".St1_Table1, out1 => #posTemp)
      Move(in := "AutoPositions".St2_Table2, out1 => "AutoPositions".St1_Table1)
      Move(in := #posTemp, out1 => "AutoPositions".St2_Table2)
   END_RUNG
   RUNG wire#powerrail
      Contact( "DevicesData".TurnTable.Status.DoneCW )
   END_RUNG wire#w1
   // the same network as SCL:
   IF "DevicesData".TurnTable.Status.DoneCCW OR "DevicesData".TurnTable.Status.DoneCW THEN
       #posTemp := "AutoPositions".St1_Table1;
       "AutoPositions".St1_Table1 := "AutoPositions".St2_Table2;
       "AutoPositions".St2_Table2 := #posTemp;
   END_IF;
END_REGION

REGION Network 8: Service doors 1
   RUNG wire#powerrail
      #ServiceDoors_Instance_1(iSequenceStoped := wire#w1, iButtonOpen := "iBtnOpenServiceDoors1", iButtonLock := "iBtnResetServiceDoors1", iSafetyOK := "iServiceDoorsLocked", iDoorClosed := "iServiceDoorClosed1", qStopSequence =>, qUnlock => "qServiceDoorUnlock1", qLightOpen => "qLEDDoors1Open", qLightLock => "qLEDDoors1EMG")
   END_RUNG
   RUNG wire#powerrail
      { S7_Templates := "SrcType := Int" } EQ_Contact(in1 := "ModeSelection_DB".mode.activeMode, in2 := "mode_0_not_selected")
   END_RUNG wire#w1
   RUNG wire#powerrail
      { S7_Templates := "SrcType := Int" } EQ_Contact(in1 := "ModeSelection_DB".mode.activeMode, in2 := "mode_1_manual")
   END_RUNG wire#w1
   // the same network as SCL:
   #ServiceDoors_Instance_1(iButtonOpen := "iBtnOpenServiceDoors1",   // "serviceDoor"
                           iButtonLock := "iBtnResetServiceDoors1",
                           iSequenceStoped := ("ModeSelection_DB".mode.activeMode = "mode_0_not_selected") OR ("ModeSelection_DB".mode.activeMode = "mode_1_manual"),
                           iSafetyOK := "iServiceDoorsLocked",
                           iDoorClosed := "iServiceDoorClosed1",
                           qUnlock => "qServiceDoorUnlock1",
                           qLightOpen => "qLEDDoors1Open",
                           qLightLock => "qLEDDoors1EMG");
END_REGION

